IF lrHighVacuumRefReading <>0 THEN
lrVacuumSoftRatio := INT_TO_LREAL(iVacuumSoftRange) /lrHighVacuumRefReading;
END_IF


IF iAnalogInput > (32767/10) THEN
rBuffer := INT_TO_LREAL(iZeroVacuumRefValue) - INT_TO_LREAL(iAnalogInput);
ELSE
rBuffer := INT_TO_LREAL(iZeroVacuumRefValue) - 3276;  (*zero- 0*)
END_IF

IF  lrVacuumSoftRatio <>0 THEN
rVacuumPV_kPa :=rBuffer/ lrVacuumSoftRatio;
END_IF

iVacuumPV_kPa := REAL_TO_INT (rVacuumPV_kPa);

END_FUNCTION_BLOCK

// ---- FBs/B_JKS_NewFB/FBP-Instrument/fbWeberMultiFreqCtrl.TcPOU
FUNCTION_BLOCK fbWeberMultiFreqCtrl
VAR_INPUT

	bErrorReset : BOOL;
	b2550NewFirmware : BOOL;
END_VAR

VAR_IN_OUT PERSISTENT
	DSWeberGenerator : ARRAY [1..iUSGeneratorQty] OF DS_WeberGenerator;
	iStepDelaySVns: INT;
END_VAR

VAR_OUTPUT
	bFSel1OnOff :  BOOL;
	bFSel2OnOff :  BOOL;

END_VAR

VAR PERSISTENT
	ARbFreqChangeTriggerEn : ARRAY [1..iUSGeneratorQty] OF BOOL; (*Internally activate by monitor the changes of set point*)
(*	ARiPowerAnalogInput AT %I* : ARRAY [1..iUSGeneratorQty] OF INT; (*Link to Terminal*)
	ARiPowerAnalogOutput AT %Q* : ARRAY [1..iUSGeneratorQty] OF INT; (*Link to Terminal*)
*)
(**)	bFreqSwitchingPBRE: ARRAY [1..iUSGeneratorQty] OF R_TRIG;
	ARbFreqChangeMonitoringEn : ARRAY [1..iUSGeneratorQty] OF BOOL; (*Enable monitor the changes of set point*)
	ARiCurrentFreq: ARRAY [1..iUSGeneratorQty] OF INT;
	iFreqChangeStep: INT;
	iFreqChangeTriggerSet: INT;
	ARbFreqChangeTriggerEnRE: ARRAY [1..iUSGeneratorQty] OF R_TRIG;
	tStep1DelayTimer: TON;
	tStep2DelayTimer: TON;
	tStep3DelayTimer: TON;
	tStep0DelayTimer: TON;
	iGenFL: INT;
	iFreqChangeFL: INT;
END_VAR

(*Ultrasonic Start/Stop Ctrl*)
tStep0DelayTimer(IN:=iFreqChangeStep = 0 , PT:=INT_TO_TIME(iStepDelaySVns) , Q=> , ET=> );

iGenFL := 1;

	FOR iGenFL := 1 TO iUSGeneratorQty DO

				(*Min Control - Default*)
				IF DSWeberGenerator[iGenFL].IN_lrPowerToAnalogRatio <= 0 THEN
				DSWeberGenerator[iGenFL].IN_lrPowerToAnalogRatio := 327.67;
				END_IF

				(*Ultrasonic Start/Stop Ctrl*)
				IF tStep0DelayTimer.Q THEN
					IF DSWeberGenerator[iGenFL].IN_bUltrasonicStartEn THEN
					DSWeberGenerator[iGenFL].OUT_bUltrasonicOnOff := TRUE;
					ELSE
					DSWeberGenerator[iGenFL].OUT_bUltrasonicOnOff := FALSE;
					END_IF

				END_IF


				(*MultiFreq Ctrl - Change Freq via Digital Output Control*)

				(*Monitoring Start/Stop Control*)
				IF DSWeberGenerator[iGenFL].IN_bMultiFreqEn THEN
					IF DSWeberGenerator[iGenFL].DSWeberMulFreqSwitching.bFreqRange2550En AND NOT DSWeberGenerator[iGenFL].DSWeberMulFreqSwitching.bFreqRange4080120En THEN
						IF DSWeberGenerator[iGenFL].IN_iFreqSetPoint = 25 OR DSWeberGenerator[iGenFL].IN_iFreqSetPoint = 50 THEN
						ARbFreqChangeMonitoringEn[iGenFL] := TRUE;
						END_IF
					ELSIF NOT DSWeberGenerator[iGenFL].DSWeberMulFreqSwitching.bFreqRange2550En AND DSWeberGenerator[iGenFL].DSWeberMulFreqSwitching.bFreqRange4080120En THEN
						IF DSWeberGenerator[iGenFL].IN_iFreqSetPoint = 40 OR DSWeberGenerator[iGenFL].IN_iFreqSetPoint = 80 OR DSWeberGenerator[iGenFL].IN_iFreqSetPoint = 132 THEN
						ARbFreqChangeMonitoringEn[iGenFL] := TRUE;
						END_IF
					ELSE
						ARbFreqChangeMonitoringEn[iGenFL] := FALSE;
					END_IF
				ELSE
						ARbFreqChangeMonitoringEn[iGenFL] := FALSE;
				END_IF

				IF ARbFreqChangeMonitoringEn[iGenFL] THEN

					IF DSWeberGenerator[iGenFL].IN_iFreqSetPoint <> ARiCurrentFreq[iGenFL] THEN
						ARbFreqChangeTriggerEn[iGenFL] := TRUE;
					END_IF

				ELSE
					ARbFreqChangeTriggerEn[iGenFL] := FALSE;
				END_IF


				(*Analog Output*)
				IF DSWeberGenerator[iGenFL].IN_lrAnalogOutputFineTuneRatio <= 0 THEN
				DSWeberGenerator[iGenFL].IN_lrAnalogOutputFineTuneRatio := 1;
				END_IF

				IF DSWeberGenerator[iGenFL].IN_iTargetPowerPercentSetPoint <= 0 THEN
				DSWeberGenerator[iGenFL].OUT_iPowerAnalogOutput := 0;
				ELSIF DSWeberGenerator[iGenFL].IN_lrPowerToAnalogRatio <= 0 THEN
				DSWeberGenerator[iGenFL].OUT_iPowerAnalogOutput := 0;
				ELSIF (INT_TO_LREAL(DSWeberGenerator[iGenFL].IN_iTargetPowerPercentSetPoint) * DSWeberGenerator[iGenFL].IN_lrPowerToAnalogRatio) * DSWeberGenerator[iGenFL].IN_lrAnalogOutputFineTuneRatio <=32767 THEN
					DSWeberGenerator[iGenFL].OUT_iPowerAnalogOutput := LREAL_TO_INT(INT_TO_LREAL(DSWeberGenerator[iGenFL].IN_iTargetPowerPercentSetPoint) * DSWeberGenerator[iGenFL].IN_lrPowerToAnalogRatio * DSWeberGenerator[iGenFL].IN_lrAnalogOutputFineTuneRatio);
				ELSIF (INT_TO_LREAL(DSWeberGenerator[iGenFL].IN_iTargetPowerPercentSetPoint) * DSWeberGenerator[iGenFL].IN_lrPowerToAnalogRatio * DSWeberGenerator[iGenFL].IN_lrAnalogOutputFineTuneRatio) >32767 THEN
					DSWeberGenerator[iGenFL].OUT_iPowerAnalogOutput := 32767;

				ELSE
				DSWeberGenerator[iGenFL].OUT_iPowerAnalogOutput := 0;
				END_IF


				(*ActualPowerPercentageDisplay*)

				IF DSWeberGenerator[iGenFL].IN_lrAnalogInputFineTuneRatio <= 0 THEN
				DSWeberGenerator[iGenFL].IN_lrAnalogInputFineTuneRatio := 1;
				END_IF

				IF DSWeberGenerator[iGenFL].IN_iPowerAnalogInput <= 0 THEN
				DSWeberGenerator[iGenFL].OUT_iActualPowerPercentDisplay := 0;
				ELSIF DSWeberGenerator[iGenFL].IN_lrPowerToAnalogRatio <= 0 THEN
				DSWeberGenerator[iGenFL].OUT_iActualPowerPercentDisplay := 0;
				ELSIF ((INT_TO_LREAL(DSWeberGenerator[iGenFL].IN_iPowerAnalogInput) / DSWeberGenerator[iGenFL].IN_lrPowerToAnalogRatio) )* DSWeberGenerator[iGenFL].IN_lrAnalogInputFineTuneRatio <=100 THEN
					DSWeberGenerator[iGenFL].OUT_iActualPowerPercentDisplay := LREAL_TO_INT((INT_TO_LREAL(DSWeberGenerator[iGenFL].IN_iPowerAnalogInput) / DSWeberGenerator[iGenFL].IN_lrPowerToAnalogRatio) * DSWeberGenerator[iGenFL].IN_lrAnalogInputFineTuneRatio);
				ELSIF ((INT_TO_LREAL(DSWeberGenerator[iGenFL].IN_iPowerAnalogInput) / DSWeberGenerator[iGenFL].IN_lrPowerToAnalogRatio) )* DSWeberGenerator[iGenFL].IN_lrAnalogInputFineTuneRatio >100 THEN
					DSWeberGenerator[iGenFL].OUT_iActualPowerPercentDisplay := 100;

				ELSE
				DSWeberGenerator[iGenFL].OUT_iPowerAnalogOutput := 0;
				END_IF

				(*TS - FreqSwitchingPushButtonControl*)
				bFreqSwitchingPBRE[iGenFL](CLK:=DSWeberGenerator[iGenFL].DSWeberMulFreqSwitching.bFreqSwitchingPB_TS , Q=> );

				IF NOT DSWeberGenerator[iGenFL].DSWeberMulFreqSwitching.bFreqRange2550En AND NOT DSWeberGenerator[iGenFL].DSWeberMulFreqSwitching.bFreqRange4080120En THEN
				DSWeberGenerator[iGenFL].DSWeberMulFreqSwitching.iFreqOutput_TS := 0;
				ELSIF DSWeberGenerator[iGenFL].DSWeberMulFreqSwitching.bFreqRange2550En AND DSWeberGenerator[iGenFL].DSWeberMulFreqSwitching.bFreqRange4080120En THEN
				DSWeberGenerator[iGenFL].DSWeberMulFreqSwitching.iFreqOutput_TS := 0;


				ELSIF DSWeberGenerator[iGenFL].DSWeberMulFreqSwitching.bFreqRange2550En AND NOT DSWeberGenerator[iGenFL].DSWeberMulFreqSwitching.bFreqRange4080120En THEN

					IF DSWeberGenerator[iGenFL].DSWeberMulFreqSwitching.iFreqOutput_TS <> 25 AND DSWeberGenerator[iGenFL].DSWeberMulFreqSwitching.iFreqOutput_TS <> 50 THEN
					DSWeberGenerator[iGenFL].DSWeberMulFreqSwitching.iFreqOutput_TS := 25;
					END_IF

					IF bFreqSwitchingPBRE[iGenFL].Q THEN
						IF DSWeberGenerator[iGenFL].DSWeberMulFreqSwitching.iFreqOutput_TS = 25 THEN
						DSWeberGenerator[iGenFL].DSWeberMulFreqSwitching.iFreqOutput_TS := 50;
						ELSIF DSWeberGenerator[iGenFL].DSWeberMulFreqSwitching.iFreqOutput_TS = 50 THEN
						DSWeberGenerator[iGenFL].DSWeberMulFreqSwitching.iFreqOutput_TS := 25;
						END_IF
					END_IF


				ELSIF NOT DSWeberGenerator[iGenFL].DSWeberMulFreqSwitching.bFreqRange2550En AND DSWeberGenerator[iGenFL].DSWeberMulFreqSwitching.bFreqRange4080120En THEN

					IF DSWeberGenerator[iGenFL].DSWeberMulFreqSwitching.iFreqOutput_TS <> 40 AND DSWeberGenerator[iGenFL].DSWeberMulFreqSwitching.iFreqOutput_TS <> 80 AND DSWeberGenerator[iGenFL].DSWeberMulFreqSwitching.iFreqOutput_TS <> 132  THEN
					DSWeberGenerator[iGenFL].DSWeberMulFreqSwitching.iFreqOutput_TS := 40;
					END_IF

					IF bFreqSwitchingPBRE[iGenFL].Q AND NOT DSWeberGenerator[iGenFL].DSWeberMulFreqSwitching.bDisableMultiFreq80kHz THEN
						IF DSWeberGenerator[iGenFL].DSWeberMulFreqSwitching.iFreqOutput_TS = 40 THEN
						DSWeberGenerator[iGenFL].DSWeberMulFreqSwitching.iFreqOutput_TS := 80;
						ELSIF DSWeberGenerator[iGenFL].DSWeberMulFreqSwitching.iFreqOutput_TS = 80 THEN
						DSWeberGenerator[iGenFL].DSWeberMulFreqSwitching.iFreqOutput_TS := 132;
						ELSIF DSWeberGenerator[iGenFL].DSWeberMulFreqSwitching.iFreqOutput_TS = 132 THEN
						DSWeberGenerator[iGenFL].DSWeberMulFreqSwitching.iFreqOutput_TS := 40;
						END_IF

					ELSIF bFreqSwitchingPBRE[iGenFL].Q AND DSWeberGenerator[iGenFL].DSWeberMulFreqSwitching.bDisableMultiFreq80kHz THEN
						IF DSWeberGenerator[iGenFL].DSWeberMulFreqSwitching.iFreqOutput_TS = 40 THEN
						DSWeberGenerator[iGenFL].DSWeberMulFreqSwitching.iFreqOutput_TS := 132;
						ELSIF DSWeberGenerator[iGenFL].DSWeberMulFreqSwitching.iFreqOutput_TS = 132 THEN
						DSWeberGenerator[iGenFL].DSWeberMulFreqSwitching.iFreqOutput_TS := 40;
						END_IF

					END_IF

				END_IF

	END_FOR



(*Seperate FL to control*)

IF iFreqChangeStep = 0 THEN
iFreqChangeFL := 1;
	FOR iFreqChangeFL := 1 TO iUSGeneratorQty DO

		IF ARbFreqChangeTriggerEn[iFreqChangeFL] THEN
		iFreqChangeStep := 1;
		iFreqChangeTriggerSet := iFreqChangeFL;
		iFreqChangeFL := iUSGeneratorQty +1;
		END_IF
	END_FOR
END_IF

(*******************************************************************************************)






(*Freq Change Start*)

IF iStepDelaySVns < 300 THEN
iStepDelaySVns := 300;
END_IF


(*Freq Change Sequence Start*)
tStep1DelayTimer(IN:=iFreqChangeStep=1 , PT:=INT_TO_TIME(iStepDelaySVns) , Q=> , ET=> );
tStep2DelayTimer(IN:=iFreqChangeStep=2 , PT:=INT_TO_TIME(iStepDelaySVns) , Q=> , ET=> );
tStep3DelayTimer(IN:=iFreqChangeStep=3 , PT:=INT_TO_TIME(iStepDelaySVns) , Q=> , ET=> );

CASE iFreqChangeStep OF
0:
	bFSel1OnOff := FALSE;
	bFSel2OnOff := FALSE;


1:
DSWeberGenerator[iFreqChangeTriggerSet].OUT_bUltrasonicOnOff := FALSE;

IF DSWeberGenerator[iFreqChangeTriggerSet].DSWeberMulFreqSwitching.bFreqRange2550En AND NOT b2550NewFirmware THEN

	IF DSWeberGenerator[iFreqChangeTriggerSet].IN_iFreqSetPoint = 25 THEN
	bFSel1OnOff := TRUE;
	bFSel2OnOff := FALSE;
	ELSIF DSWeberGenerator[iFreqChangeTriggerSet].IN_iFreqSetPoint = 50 THEN
	bFSel1OnOff := FALSE;
	bFSel2OnOff := TRUE;
	ELSIF DSWeberGenerator[iFreqChangeTriggerSet].IN_iFreqSetPoint = 0 THEN
	bFSel1OnOff := FALSE;
	bFSel2OnOff := FALSE;
	ELSE
	bFSel1OnOff := FALSE;
	bFSel2OnOff := FALSE;
	iFreqChangeStep := 4;
	END_IF

ELSIF DSWeberGenerator[iFreqChangeTriggerSet].DSWeberMulFreqSwitching.bFreqRange2550En AND b2550NewFirmware THEN

	IF DSWeberGenerator[iFreqChangeTriggerSet].IN_iFreqSetPoint = 25 THEN
	bFSel1OnOff := TRUE;
	bFSel2OnOff := TRUE;
	ELSIF DSWeberGenerator[iFreqChangeTriggerSet].IN_iFreqSetPoint = 50 THEN
	bFSel1OnOff := FALSE;
	bFSel2OnOff := TRUE;
	ELSIF DSWeberGenerator[iFreqChangeTriggerSet].IN_iFreqSetPoint = 0 THEN
	bFSel1OnOff := FALSE;
	bFSel2OnOff := FALSE;
	ELSE
	bFSel1OnOff := FALSE;
	bFSel2OnOff := FALSE;
	iFreqChangeStep := 4;
	END_IF

END_IF

IF DSWeberGenerator[iFreqChangeTriggerSet].DSWeberMulFreqSwitching.bFreqRange4080120En THEN

	IF NOT DSWeberGenerator[iFreqChangeTriggerSet].DSWeberMulFreqSwitching.bDisableMultiFreq80kHz THEN

			IF DSWeberGenerator[iFreqChangeTriggerSet].IN_iFreqSetPoint = 40 THEN
			bFSel1OnOff := TRUE;
			bFSel2OnOff := TRUE;
			ELSIF DSWeberGenerator[iFreqChangeTriggerSet].IN_iFreqSetPoint = 80 THEN
			bFSel1OnOff := FALSE;
			bFSel2OnOff := TRUE;
			ELSIF DSWeberGenerator[iFreqChangeTriggerSet].IN_iFreqSetPoint = 132 THEN
			bFSel1OnOff := TRUE;
			bFSel2OnOff := FALSE;
			ELSIF DSWeberGenerator[iFreqChangeTriggerSet].IN_iFreqSetPoint = 0 THEN
			bFSel1OnOff := FALSE;
			bFSel2OnOff := FALSE;
			ELSE
			bFSel1OnOff := FALSE;
			bFSel2OnOff := FALSE;
			iFreqChangeStep := 4;
			END_IF
	ELSE

			IF DSWeberGenerator[iFreqChangeTriggerSet].IN_iFreqSetPoint = 40 THEN
			bFSel1OnOff := TRUE;
			bFSel2OnOff := FALSE;
			ELSIF DSWeberGenerator[iFreqChangeTriggerSet].IN_iFreqSetPoint = 132 THEN
			bFSel1OnOff := FALSE;
			bFSel2OnOff := TRUE;
			ELSIF DSWeberGenerator[iFreqChangeTriggerSet].IN_iFreqSetPoint = 0 THEN
			bFSel1OnOff := FALSE;
			bFSel2OnOff := FALSE;
			ELSE
			bFSel1OnOff := FALSE;
			bFSel2OnOff := FALSE;
			iFreqChangeStep := 4;
			END_IF
	END_IF



END_IF


IF tStep1DelayTimer.Q THEN
iFreqChangeStep := 2;
END_IF

2:
IF DSWeberGenerator[iFreqChangeTriggerSet].IN_iFreqSetPoint <> 0 THEN
DSWeberGenerator[iFreqChangeTriggerSet].OUT_bUltrasonicOnOff := TRUE;
ELSE
DSWeberGenerator[iFreqChangeTriggerSet].OUT_bUltrasonicOnOff := FALSE;
END_IF

IF tStep2DelayTimer.Q THEN
iFreqChangeStep := 3;
END_IF

3:
DSWeberGenerator[iFreqChangeTriggerSet].OUT_bUltrasonicOnOff := FALSE;
bFSel1OnOff := FALSE;
bFSel2OnOff := FALSE;

IF tStep3DelayTimer.Q THEN
iFreqChangeStep := 0;
ARbFreqChangeTriggerEn[iFreqChangeTriggerSet] := FALSE;
ARiCurrentFreq[iFreqChangeTriggerSet] := DSWeberGenerator[iFreqChangeTriggerSet].IN_iFreqSetPoint;
END_IF

4: (*Error*)
DSWeberGenerator[iFreqChangeTriggerSet].OUT_bFreqSetPointError := TRUE;
iFreqChangeStep := 5;


5: (*Error - Waiting Reset*)
IF bErrorReset THEN
DSWeberGenerator[iFreqChangeTriggerSet].OUT_bFreqSetPointError := FALSE;
iFreqChangeStep := 0;
ARbFreqChangeTriggerEn[iFreqChangeTriggerSet] := FALSE;
ARiCurrentFreq[iFreqChangeTriggerSet] := DSWeberGenerator[iFreqChangeTriggerSet].IN_iFreqSetPoint;
END_IF

END_CASE

END_FUNCTION_BLOCK

// ---- FBs/B_JKS_NewFB/FBP-Instrument/fbBrensonMultiFreqCtrl.TcPOU
FUNCTION_BLOCK fbBrensonMultiFreqCtrl
VAR_INPUT

	bErrorReset : BOOL;
	b2550NewFirmware : BOOL;
END_VAR

VAR_IN_OUT PERSISTENT
	DSBrensonGenerator : ARRAY [1..iUSGeneratorQty] OF DS_BrensonGenerator;
	iStepDelaySVns: INT;
END_VAR

VAR_OUTPUT
	bFSel1OnOff :  BOOL;
	bFSel2OnOff :  BOOL;

END_VAR

VAR PERSISTENT
	ARbFreqChangeTriggerEn : ARRAY [1..iUSGeneratorQty] OF BOOL; (*Internally activate by monitor the changes of set point*)
(*	ARiPowerAnalogInput AT %I* : ARRAY [1..iUSGeneratorQty] OF INT; (*Link to Terminal*)
	ARiPowerAnalogOutput AT %Q* : ARRAY [1..iUSGeneratorQty] OF INT; (*Link to Terminal*)
*)
(**)	bFreqSwitchingPBRE: ARRAY [1..iUSGeneratorQty] OF R_TRIG;
	ARbFreqChangeMonitoringEn : ARRAY [1..iUSGeneratorQty] OF BOOL; (*Enable monitor the changes of set point*)
	ARiCurrentFreq: ARRAY [1..iUSGeneratorQty] OF INT;
	iFreqChangeStep: INT;
	iFreqChangeTriggerSet: INT;
	ARbFreqChangeTriggerEnRE: ARRAY [1..iUSGeneratorQty] OF R_TRIG;
	tStep1DelayTimer: TON;
	tStep2DelayTimer: TON;
	tStep3DelayTimer: TON;
	tStep0DelayTimer: TON;
	iGenFL: INT;
	iFreqChangeFL: INT;
END_VAR

(*Ultrasonic Start/Stop Ctrl*)
tStep0DelayTimer(IN:=iFreqChangeStep = 0 , PT:=INT_TO_TIME(iStepDelaySVns) , Q=> , ET=> );

iGenFL := 1;

	FOR iGenFL := 1 TO iUSGeneratorQty DO

				(*Min Control - Default*)
				IF DSBrensonGenerator[iGenFL].IN_lrPowerToAnalogRatio <= 0 THEN
				DSBrensonGenerator[iGenFL].IN_lrPowerToAnalogRatio := 327.67;
				END_IF

				(*Ultrasonic Start/Stop Ctrl*)
				IF tStep0DelayTimer.Q THEN
					IF DSBrensonGenerator[iGenFL].IN_bUltrasonicStartEn THEN
					DSBrensonGenerator[iGenFL].OUT_bUltrasonicOnOff := TRUE;
					ELSE
					DSBrensonGenerator[iGenFL].OUT_bUltrasonicOnOff := FALSE;
					END_IF

				END_IF


				(*MultiFreq Ctrl - Change Freq via Digital Output Control*)

				(*Monitoring Start/Stop Control*)
				IF DSBrensonGenerator[iGenFL].IN_bMultiFreqEn THEN
					IF DSBrensonGenerator[iGenFL].DSBrensonMulFreqSwitching.bFreqRange2550En AND NOT DSBrensonGenerator[iGenFL].DSBrensonMulFreqSwitching.bFreqRange4080120En THEN
						IF DSBrensonGenerator[iGenFL].IN_iFreqSetPoint = 25 OR DSBrensonGenerator[iGenFL].IN_iFreqSetPoint = 50 THEN
						ARbFreqChangeMonitoringEn[iGenFL] := TRUE;
						END_IF
					ELSIF NOT DSBrensonGenerator[iGenFL].DSBrensonMulFreqSwitching.bFreqRange2550En AND DSBrensonGenerator[iGenFL].DSBrensonMulFreqSwitching.bFreqRange4080120En THEN
						IF DSBrensonGenerator[iGenFL].IN_iFreqSetPoint = 40 OR DSBrensonGenerator[iGenFL].IN_iFreqSetPoint = 80 OR DSBrensonGenerator[iGenFL].IN_iFreqSetPoint = 120 THEN
						ARbFreqChangeMonitoringEn[iGenFL] := TRUE;
						END_IF
					ELSE
						ARbFreqChangeMonitoringEn[iGenFL] := FALSE;
					END_IF
				ELSE
						ARbFreqChangeMonitoringEn[iGenFL] := FALSE;
				END_IF

				IF ARbFreqChangeMonitoringEn[iGenFL] THEN

					IF DSBrensonGenerator[iGenFL].IN_iFreqSetPoint <> ARiCurrentFreq[iGenFL] THEN
						ARbFreqChangeTriggerEn[iGenFL] := TRUE;
					END_IF

				ELSE
					ARbFreqChangeTriggerEn[iGenFL] := FALSE;
				END_IF


				(*Analog Output*)
				IF DSBrensonGenerator[iGenFL].IN_lrAnalogOutputFineTuneRatio <= 0 THEN
				DSBrensonGenerator[iGenFL].IN_lrAnalogOutputFineTuneRatio := 1;
				END_IF

				IF DSBrensonGenerator[iGenFL].IN_iTargetPowerPercentSetPoint <= 0 THEN
				DSBrensonGenerator[iGenFL].OUT_iPowerAnalogOutput := 0;
				ELSIF DSBrensonGenerator[iGenFL].IN_lrPowerToAnalogRatio <= 0 THEN
				DSBrensonGenerator[iGenFL].OUT_iPowerAnalogOutput := 0;
				ELSIF (INT_TO_LREAL(DSBrensonGenerator[iGenFL].IN_iTargetPowerPercentSetPoint) * DSBrensonGenerator[iGenFL].IN_lrPowerToAnalogRatio) * DSBrensonGenerator[iGenFL].IN_lrAnalogOutputFineTuneRatio <=32767 THEN
					DSBrensonGenerator[iGenFL].OUT_iPowerAnalogOutput := LREAL_TO_INT(INT_TO_LREAL(DSBrensonGenerator[iGenFL].IN_iTargetPowerPercentSetPoint) * DSBrensonGenerator[iGenFL].IN_lrPowerToAnalogRatio * DSBrensonGenerator[iGenFL].IN_lrAnalogOutputFineTuneRatio);
				ELSIF (INT_TO_LREAL(DSBrensonGenerator[iGenFL].IN_iTargetPowerPercentSetPoint) * DSBrensonGenerator[iGenFL].IN_lrPowerToAnalogRatio * DSBrensonGenerator[iGenFL].IN_lrAnalogOutputFineTuneRatio) >32767 THEN
					DSBrensonGenerator[iGenFL].OUT_iPowerAnalogOutput := 32767;

				ELSE
				DSBrensonGenerator[iGenFL].OUT_iPowerAnalogOutput := 0;
				END_IF


				(*ActualPowerPercentageDisplay*)

				IF DSBrensonGenerator[iGenFL].IN_lrAnalogInputFineTuneRatio <= 0 THEN
				DSBrensonGenerator[iGenFL].IN_lrAnalogInputFineTuneRatio := 1;
				END_IF

				IF DSBrensonGenerator[iGenFL].IN_iPowerAnalogInput <= 0 THEN
				DSBrensonGenerator[iGenFL].OUT_iActualPowerPercentDisplay := 0;
				ELSIF DSBrensonGenerator[iGenFL].IN_lrPowerToAnalogRatio <= 0 THEN
				DSBrensonGenerator[iGenFL].OUT_iActualPowerPercentDisplay := 0;
				ELSIF ((INT_TO_LREAL(DSBrensonGenerator[iGenFL].IN_iPowerAnalogInput) / DSBrensonGenerator[iGenFL].IN_lrPowerToAnalogRatio) )* DSBrensonGenerator[iGenFL].IN_lrAnalogInputFineTuneRatio <=100 THEN
					DSBrensonGenerator[iGenFL].OUT_iActualPowerPercentDisplay := LREAL_TO_INT((INT_TO_LREAL(DSBrensonGenerator[iGenFL].IN_iPowerAnalogInput) / DSBrensonGenerator[iGenFL].IN_lrPowerToAnalogRatio) * DSBrensonGenerator[iGenFL].IN_lrAnalogInputFineTuneRatio);
				ELSIF ((INT_TO_LREAL(DSBrensonGenerator[iGenFL].IN_iPowerAnalogInput) / DSBrensonGenerator[iGenFL].IN_lrPowerToAnalogRatio) )* DSBrensonGenerator[iGenFL].IN_lrAnalogInputFineTuneRatio >100 THEN
					DSBrensonGenerator[iGenFL].OUT_iActualPowerPercentDisplay := 100;

				ELSE
				DSBrensonGenerator[iGenFL].OUT_iPowerAnalogOutput := 0;
				END_IF

				(*TS - FreqSwitchingPushButtonControl*)
				bFreqSwitchingPBRE[iGenFL](CLK:=DSBrensonGenerator[iGenFL].DSBrensonMulFreqSwitching.bFreqSwitchingPB_TS , Q=> );

				IF NOT DSBrensonGenerator[iGenFL].DSBrensonMulFreqSwitching.bFreqRange2550En AND NOT DSBrensonGenerator[iGenFL].DSBrensonMulFreqSwitching.bFreqRange4080120En THEN
				DSBrensonGenerator[iGenFL].DSBrensonMulFreqSwitching.iFreqOutput_TS := 0;
				ELSIF DSBrensonGenerator[iGenFL].DSBrensonMulFreqSwitching.bFreqRange2550En AND DSBrensonGenerator[iGenFL].DSBrensonMulFreqSwitching.bFreqRange4080120En THEN
				DSBrensonGenerator[iGenFL].DSBrensonMulFreqSwitching.iFreqOutput_TS := 0;


				ELSIF DSBrensonGenerator[iGenFL].DSBrensonMulFreqSwitching.bFreqRange2550En AND NOT DSBrensonGenerator[iGenFL].DSBrensonMulFreqSwitching.bFreqRange4080120En THEN

					IF DSBrensonGenerator[iGenFL].DSBrensonMulFreqSwitching.iFreqOutput_TS <> 25 AND DSBrensonGenerator[iGenFL].DSBrensonMulFreqSwitching.iFreqOutput_TS <> 50 THEN
					DSBrensonGenerator[iGenFL].DSBrensonMulFreqSwitching.iFreqOutput_TS := 25;
					END_IF

					IF bFreqSwitchingPBRE[iGenFL].Q THEN
						IF DSBrensonGenerator[iGenFL].DSBrensonMulFreqSwitching.iFreqOutput_TS = 25 THEN
						DSBrensonGenerator[iGenFL].DSBrensonMulFreqSwitching.iFreqOutput_TS := 50;
						ELSIF DSBrensonGenerator[iGenFL].DSBrensonMulFreqSwitching.iFreqOutput_TS = 50 THEN
						DSBrensonGenerator[iGenFL].DSBrensonMulFreqSwitching.iFreqOutput_TS := 25;
						END_IF
					END_IF


				ELSIF NOT DSBrensonGenerator[iGenFL].DSBrensonMulFreqSwitching.bFreqRange2550En AND DSBrensonGenerator[iGenFL].DSBrensonMulFreqSwitching.bFreqRange4080120En THEN

					IF DSBrensonGenerator[iGenFL].DSBrensonMulFreqSwitching.iFreqOutput_TS <> 40 AND DSBrensonGenerator[iGenFL].DSBrensonMulFreqSwitching.iFreqOutput_TS <> 80 AND DSBrensonGenerator[iGenFL].DSBrensonMulFreqSwitching.iFreqOutput_TS <> 120  THEN
					DSBrensonGenerator[iGenFL].DSBrensonMulFreqSwitching.iFreqOutput_TS := 40;
					END_IF

					IF bFreqSwitchingPBRE[iGenFL].Q AND NOT DSBrensonGenerator[iGenFL].DSBrensonMulFreqSwitching.bDisableMultiFreq80kHz THEN
						IF DSBrensonGenerator[iGenFL].DSBrensonMulFreqSwitching.iFreqOutput_TS = 40 THEN
						DSBrensonGenerator[iGenFL].DSBrensonMulFreqSwitching.iFreqOutput_TS := 80;
						ELSIF DSBrensonGenerator[iGenFL].DSBrensonMulFreqSwitching.iFreqOutput_TS = 80 THEN
						DSBrensonGenerator[iGenFL].DSBrensonMulFreqSwitching.iFreqOutput_TS := 120;
						ELSIF DSBrensonGenerator[iGenFL].DSBrensonMulFreqSwitching.iFreqOutput_TS = 120 THEN
						DSBrensonGenerator[iGenFL].DSBrensonMulFreqSwitching.iFreqOutput_TS := 40;
						END_IF

					ELSIF bFreqSwitchingPBRE[iGenFL].Q AND DSBrensonGenerator[iGenFL].DSBrensonMulFreqSwitching.bDisableMultiFreq80kHz THEN
						IF DSBrensonGenerator[iGenFL].DSBrensonMulFreqSwitching.iFreqOutput_TS = 40 THEN
						DSBrensonGenerator[iGenFL].DSBrensonMulFreqSwitching.iFreqOutput_TS := 120;
						ELSIF DSBrensonGenerator[iGenFL].DSBrensonMulFreqSwitching.iFreqOutput_TS = 120 THEN
						DSBrensonGenerator[iGenFL].DSBrensonMulFreqSwitching.iFreqOutput_TS := 40;
						END_IF

					END_IF

				END_IF

	END_FOR



(*Seperate FL to control*)

IF iFreqChangeStep = 0 THEN
iFreqChangeFL := 1;
	FOR iFreqChangeFL := 1 TO iUSGeneratorQty DO

		IF ARbFreqChangeTriggerEn[iFreqChangeFL] THEN
		iFreqChangeStep := 1;
		iFreqChangeTriggerSet := iFreqChangeFL;
		iFreqChangeFL := iUSGeneratorQty +1;
		END_IF
	END_FOR
END_IF

(*******************************************************************************************)






(*Freq Change Start*)

IF iStepDelaySVns < 300 THEN
iStepDelaySVns := 300;
END_IF


(*Freq Change Sequence Start*)
tStep1DelayTimer(IN:=iFreqChangeStep=1 , PT:=INT_TO_TIME(iStepDelaySVns) , Q=> , ET=> );
tStep2DelayTimer(IN:=iFreqChangeStep=2 , PT:=INT_TO_TIME(iStepDelaySVns) , Q=> , ET=> );
tStep3DelayTimer(IN:=iFreqChangeStep=3 , PT:=INT_TO_TIME(iStepDelaySVns) , Q=> , ET=> );

CASE iFreqChangeStep OF
0:
	bFSel1OnOff := FALSE;
	bFSel2OnOff := FALSE;


1:
DSBrensonGenerator[iFreqChangeTriggerSet].OUT_bUltrasonicOnOff := FALSE;

IF DSBrensonGenerator[iFreqChangeTriggerSet].DSBrensonMulFreqSwitching.bFreqRange2550En AND NOT b2550NewFirmware THEN

	IF DSBrensonGenerator[iFreqChangeTriggerSet].IN_iFreqSetPoint = 25 THEN
	bFSel1OnOff := TRUE;
	bFSel2OnOff := FALSE;
	ELSIF DSBrensonGenerator[iFreqChangeTriggerSet].IN_iFreqSetPoint = 50 THEN
	bFSel1OnOff := FALSE;
	bFSel2OnOff := TRUE;
	ELSIF DSBrensonGenerator[iFreqChangeTriggerSet].IN_iFreqSetPoint = 0 THEN
	bFSel1OnOff := FALSE;
	bFSel2OnOff := FALSE;
	ELSE
	bFSel1OnOff := FALSE;
	bFSel2OnOff := FALSE;
	iFreqChangeStep := 4;
	END_IF

ELSIF DSBrensonGenerator[iFreqChangeTriggerSet].DSBrensonMulFreqSwitching.bFreqRange2550En AND b2550NewFirmware THEN

	IF DSBrensonGenerator[iFreqChangeTriggerSet].IN_iFreqSetPoint = 25 THEN
	bFSel1OnOff := TRUE;
	bFSel2OnOff := TRUE;
	ELSIF DSBrensonGenerator[iFreqChangeTriggerSet].IN_iFreqSetPoint = 50 THEN
	bFSel1OnOff := FALSE;
	bFSel2OnOff := TRUE;
	ELSIF DSBrensonGenerator[iFreqChangeTriggerSet].IN_iFreqSetPoint = 0 THEN
	bFSel1OnOff := FALSE;
	bFSel2OnOff := FALSE;
	ELSE
	bFSel1OnOff := FALSE;
	bFSel2OnOff := FALSE;
	iFreqChangeStep := 4;
	END_IF

END_IF

IF DSBrensonGenerator[iFreqChangeTriggerSet].DSBrensonMulFreqSwitching.bFreqRange4080120En THEN

	IF NOT DSBrensonGenerator[iFreqChangeTriggerSet].DSBrensonMulFreqSwitching.bDisableMultiFreq80kHz THEN

			IF DSBrensonGenerator[iFreqChangeTriggerSet].IN_iFreqSetPoint = 40 THEN
			bFSel1OnOff := TRUE;
			bFSel2OnOff := TRUE;
			ELSIF DSBrensonGenerator[iFreqChangeTriggerSet].IN_iFreqSetPoint = 80 THEN
			bFSel1OnOff := FALSE;
			bFSel2OnOff := TRUE;
			ELSIF DSBrensonGenerator[iFreqChangeTriggerSet].IN_iFreqSetPoint = 120 THEN
			bFSel1OnOff := TRUE;
			bFSel2OnOff := FALSE;
			ELSIF DSBrensonGenerator[iFreqChangeTriggerSet].IN_iFreqSetPoint = 0 THEN
			bFSel1OnOff := FALSE;
			bFSel2OnOff := FALSE;
			ELSE
			bFSel1OnOff := FALSE;
			bFSel2OnOff := FALSE;
			iFreqChangeStep := 4;
			END_IF
	ELSE

			IF DSBrensonGenerator[iFreqChangeTriggerSet].IN_iFreqSetPoint = 40 THEN
			bFSel1OnOff := TRUE;
			bFSel2OnOff := FALSE;
			ELSIF DSBrensonGenerator[iFreqChangeTriggerSet].IN_iFreqSetPoint = 120 THEN
			bFSel1OnOff := FALSE;
			bFSel2OnOff := TRUE;
			ELSIF DSBrensonGenerator[iFreqChangeTriggerSet].IN_iFreqSetPoint = 0 THEN
			bFSel1OnOff := FALSE;
			bFSel2OnOff := FALSE;
			ELSE
			bFSel1OnOff := FALSE;
			bFSel2OnOff := FALSE;
			iFreqChangeStep := 4;
			END_IF
	END_IF



END_IF


IF tStep1DelayTimer.Q THEN
iFreqChangeStep := 2;
END_IF

2:
IF DSBrensonGenerator[iFreqChangeTriggerSet].IN_iFreqSetPoint <> 0 THEN
DSBrensonGenerator[iFreqChangeTriggerSet].OUT_bUltrasonicOnOff := TRUE;
ELSE
DSBrensonGenerator[iFreqChangeTriggerSet].OUT_bUltrasonicOnOff := FALSE;
END_IF

IF tStep2DelayTimer.Q THEN
iFreqChangeStep := 3;
END_IF

3:
DSBrensonGenerator[iFreqChangeTriggerSet].OUT_bUltrasonicOnOff := FALSE;
bFSel1OnOff := FALSE;
bFSel2OnOff := FALSE;

IF tStep3DelayTimer.Q THEN
iFreqChangeStep := 0;
ARbFreqChangeTriggerEn[iFreqChangeTriggerSet] := FALSE;
ARiCurrentFreq[iFreqChangeTriggerSet] := DSBrensonGenerator[iFreqChangeTriggerSet].IN_iFreqSetPoint;
END_IF

4: (*Error*)
DSBrensonGenerator[iFreqChangeTriggerSet].OUT_bFreqSetPointError := TRUE;
iFreqChangeStep := 5;


5: (*Error - Waiting Reset*)
IF bErrorReset THEN
DSBrensonGenerator[iFreqChangeTriggerSet].OUT_bFreqSetPointError := FALSE;
iFreqChangeStep := 0;
ARbFreqChangeTriggerEn[iFreqChangeTriggerSet] := FALSE;
ARiCurrentFreq[iFreqChangeTriggerSet] := DSBrensonGenerator[iFreqChangeTriggerSet].IN_iFreqSetPoint;
END_IF

END_CASE

END_FUNCTION_BLOCK

// ---- FBs/B_JKS_CustomFB/fbBarcodeCtrl/fbBarcodeTracer.TcPOU
FUNCTION_BLOCK fbBarcodeTracer
VAR_INPUT
	bTracerST : BOOL;
	sTargetBarcode : STRING;
	AR99sBarCodeRaw : ARRAY [0..iProductRecipeArrayQty] OF STRING;
	AR99sBarcodeDescrip	: ARRAY [0..iProductRecipeArrayQty] OF STRING;


END_VAR
VAR_OUTPUT

	bBarcodeTraceSuccess : BOOL;
	bBarcodeTraceFail : BOOL;
	iBarcodeInRecipeNo : INT;
	sBarcodeInDescrip	: STRING;
END_VAR
VAR
	i: INT;
	TracerRE : R_TRIG;

	sBuffer: STRING;
	STEP: INT;
END_VAR

TracerRE(CLK:=bTracerST,Q=>);

IF NOT bTracerST THEN
	bBarcodeTraceSuccess := FALSE;
	bBarcodeTraceFail := FALSE;
	iBarcodeInRecipeNo := 0;
	i := 1;
END_IF

IF bTracerST AND sTargetBarcode <> '' (*AND sTargetBarcode <> sBuffer*) THEN

		(*sBuffer := sTargetBarcode;*)
		FOR i := 1 TO 99 DO

		IF sTargetBarcode = AR99sBarCodeRaw[i] THEN
		sBarcodeInDescrip := AR99sBarcodeDescrip[i];
		iBarcodeInRecipeNo := i;
		bBarcodeTraceSuccess := TRUE;
		(*bBarcodeTraceFail := FALSE;*)
		i := 100;
		(*ELSE
		bBarcodeTraceFail := TRUE;
		bBarcodeTraceSuccess := FALSE;*)
		END_IF

		END_FOR

END_IF
IF (i > 99 AND bTracerST AND NOT bBarcodeTraceSuccess) (*OR (sTargetBarcode = '')*) THEN
bBarcodeTraceFail := TRUE;
ELSE
bBarcodeTraceFail := FALSE;
END_IF

END_FUNCTION_BLOCK

// ---- FBs/B_JKS_CustomFB/fbBarcodeCtrl/fbPreSuffixEliminator.TcPOU
FUNCTION_BLOCK fbPreSuffixEliminator
VAR_INPUT
	bEN									: BOOL;
	bPrefixEliminatorEN					: BOOL;
	bSuffixEliminatorEN					: BOOL;
	sData								: STRING;
	sPrefix								: STRING (*:='$02'*);
	sSuffix								:STRING;
	iLengthAfterPrefix						: INT;
	iLengthBeforeSuffix					: INT;

END_VAR
VAR_OUTPUT

	sPrefixEliminatorResult					: STRING;
	sSuffixEliminatorResult					: STRING;
	sPreSuffixEliminatorResult				: STRING;
	sNoneEliminatorReseult				: STRING;

END_VAR
VAR
	iBCPrefixFound						: INT;
	iBCSuffixFound						: INT;
	sIntPrefixEliminatorResult				: STRING;
END_VAR

(*Prefix Eliminator*)
IF bEN AND bPrefixEliminatorEN AND NOT bSuffixEliminatorEN THEN

sSuffixEliminatorResult := '';
sPreSuffixEliminatorResult := '';

iBCPrefixFound:=FIND(sData, sPrefix);
sPrefixEliminatorResult:=RIGHT(sData, iBCPrefixFound+iLengthAfterPrefix);

END_IF

(*Suffix Eliminator*)
IF bEN AND bSuffixEliminatorEN AND NOT bPrefixEliminatorEN THEN

sPrefixEliminatorResult := '';
sPreSuffixEliminatorResult := '';


iBCSuffixFound:=FIND(sData, sSuffix);
sSuffixEliminatorResult:=LEFT(sData, iBCSuffixFound-iLengthBeforeSuffix);

END_IF



IF bEN AND bSuffixEliminatorEN AND bPrefixEliminatorEN THEN

sPrefixEliminatorResult := '';
sSuffixEliminatorResult := '';

iBCPrefixFound:=FIND(sData, sPrefix);
sIntPrefixEliminatorResult:=RIGHT(sData, iBCPrefixFound+iLengthAfterPrefix);


iBCSuffixFound:=FIND(sIntPrefixEliminatorResult, sSuffix);
sPreSuffixEliminatorResult:=LEFT(sIntPrefixEliminatorResult, iBCSuffixFound-iLengthBeforeSuffix);

END_IF



IF bEN AND NOT bSuffixEliminatorEN AND NOT bPrefixEliminatorEN THEN

sNoneEliminatorReseult:=sData;

END_IF

END_FUNCTION_BLOCK

// ---- FBs/B_JKS_CustomFB/fbBarcodeCtrl/fbBarcodeSorting_10ML5575.TcPOU
FUNCTION_BLOCK fbBarcodeSorting_10ML5575
VAR_INPUT
	bEN : BOOL;
	bBarcodeTracerInvalidFlag : BOOL;
	bConfirmPB : BOOL;

	ARbBarcodeStorageEnable : ARRAY [0..10] OF BOOL;

END_VAR
VAR_IN_OUT
	sBarcodeInputFromScanner : STRING;
	ARbHMIBarcodeScanEn : ARRAY [0..10] OF BOOL;
	ARsHMIBarcodeData_ScanIn : ARRAY [0..10] OF STRING(50);


	(*Result for Out after Confirm button press*)
	ARsBarcodeData_LdBasketInfo : ARRAY [0..10] OF STRING(50);

END_VAR

VAR_OUTPUT
	bBarcodeScanEnableFlag : BOOL;
	bConfirmReadyFlag : BOOL;
END_VAR
VAR

	ARbHMIBarcodeScanEnRE: ARRAY [0..10] OF R_TRIG;
	iREFL: INT;
	iREFL2: INT;
	iScanFL: INT;
	iConfirmFL: INT;
	ARsHMIBarcodeData_Empty : ARRAY [0..10] OF STRING(50);
	bConfirmPBRE: R_TRIG;
END_VAR

bConfirmPBRE(CLK:= bConfirmPB, Q=> );


iREFL := 1;
FOR iREFL := 1 TO 10 DO
	IF iREFL >= 1 AND iREFL <= 10 THEN
		ARbHMIBarcodeScanEnRE[iREFL](CLK:=ARbHMIBarcodeScanEn[iREFL] , Q=> );

		IF ARbHMIBarcodeScanEnRE[iREFL].Q THEN
			iREFL2 := 1;

			FOR iREFL2 := 1 TO 10 DO
				ARbHMIBarcodeScanEn[iREFL2] := FALSE;
			END_FOR

			ARbHMIBarcodeScanEn[iREFL] := TRUE;
			bBarcodeScanEnableFlag := TRUE;
		END_IF
	END_IF

END_FOR

iScanFL := 1;
FOR iScanFL := 1 TO 10 DO
	IF iScanFL >= 1 AND iScanFL <= 10 THEN


		IF ARbBarcodeStorageEnable[iScanFL] (*AND ARbHMIBarcodeScanEn[iScanFL] *) AND sBarcodeInputFromScanner <> '' THEN
			ARsHMIBarcodeData_ScanIn[iScanFL]	:= sBarcodeInputFromScanner;
			bBarcodeScanEnableFlag 				:= FALSE;
			ARbHMIBarcodeScanEn[iScanFL] 		:= FALSE;
			(*sBarcodeInputFromScanner			:= '';*)
		END_IF
	END_IF
END_FOR

iConfirmFL := 1;
bConfirmReadyFlag := TRUE;

IF bBarcodeTracerInvalidFlag THEN
bConfirmReadyFlag := FALSE;
END_IF

FOR iConfirmFL := 1 TO 10 DO
	IF iConfirmFL >= 1 AND iConfirmFL <= 10 THEN
		IF ARbBarcodeStorageEnable[iConfirmFL] AND ARsHMIBarcodeData_ScanIn[iConfirmFL] = '' THEN
		bConfirmReadyFlag := FALSE;
		END_IF
	END_IF
END_FOR


IF bConfirmPBRE.Q AND bConfirmReadyFlag THEN
ARsBarcodeData_LdBasketInfo 	:= ARsHMIBarcodeData_ScanIn;
ARsHMIBarcodeData_ScanIn 	:= ARsHMIBarcodeData_Empty ;
END_IF


IF NOT bEN THEN
ARsHMIBarcodeData_ScanIn 	:= ARsHMIBarcodeData_Empty ;
END_IF

END_FUNCTION_BLOCK

// ---- FBs/B_JKS_NewFB_V2/FBP-BasketInfoRelated/fbV2_BasketInfoManager.TcPOU
FUNCTION_BLOCK fbV2_BasketInfoManager
VAR_INPUT
	iRecipeChangeFlagDelayTime_Sec : REAL;
END_VAR
VAR_OUTPUT
	bRecipeChangedFlag : BOOL;
	bMinMaxEffChangeFlag : BOOL;

END_VAR
VAR_IN_OUT
	DSV2BasketInfo : DSV2_BasketInfo;
END_VAR

VAR
	tRecipeChangeFlagDelayOffTimer: TON;
	DSV2BasketInfoEmpty : DSV2_BasketInfo;

	iPRNBuffer: INT;
	tMinMaxEffChangeDelayOffTimer: TON;
	iFL: INT;
END_VAR

VAR PERSISTENT
	iPreviousProductRecipeNo: INT;
	ARiCurrentData : ARRAY [1..20] OF INT;
	ARiPreviousData : ARRAY [1..20] OF INT;

END_VAR

(*bMinMaxEffChangeFlag Control*)
ARiCurrentData[1] := DSV2BasketInfo.iCurrentStationNo;
ARiCurrentData[2] := DSV2BasketInfo.iPreviousStationNo;
ARiCurrentData[3] := DSV2BasketInfo.iProductRecipeStepNo;
ARiCurrentData[4] := DSV2BasketInfo.iStationSeqenceRecipeNo;
ARiCurrentData[5] := 0;

ARiCurrentData[6] := DSV2BasketInfo.DSV2MinMaxEffTime.ARiEffTime[1];
ARiCurrentData[7] := DSV2BasketInfo.DSV2MinMaxEffTime.ARiMaxTime[1];
ARiCurrentData[8] := DSV2BasketInfo.DSV2MinMaxEffTime.ARiMinTime[1];
ARiCurrentData[9] := DSV2BasketInfo.DSV2MinMaxEffTime.ARiStnSeqRepNo[1];
ARiCurrentData[10] := DSV2BasketInfo.DSV2MinMaxEffTime.ARiTransferStationNo[1];

ARiCurrentData[11] := DSV2BasketInfo.DSV2MinMaxEffTime.ARiEffTime[2];
ARiCurrentData[12] := DSV2BasketInfo.DSV2MinMaxEffTime.ARiMaxTime[2];
ARiCurrentData[13] := DSV2BasketInfo.DSV2MinMaxEffTime.ARiMinTime[2];
ARiCurrentData[14] := DSV2BasketInfo.DSV2MinMaxEffTime.ARiStnSeqRepNo[2];
ARiCurrentData[15] := DSV2BasketInfo.DSV2MinMaxEffTime.ARiTransferStationNo[2];

ARiCurrentData[16] := DSV2BasketInfo.DSV2MinMaxEffTime.ARiEffTime[3];
ARiCurrentData[17] := DSV2BasketInfo.DSV2MinMaxEffTime.ARiMaxTime[3];
ARiCurrentData[18] := DSV2BasketInfo.DSV2MinMaxEffTime.ARiMinTime[3];
ARiCurrentData[19] := DSV2BasketInfo.DSV2MinMaxEffTime.ARiStnSeqRepNo[3];
ARiCurrentData[20] := DSV2BasketInfo.DSV2MinMaxEffTime.ARiTransferStationNo[3];



iFL := 1;
	FOR iFL := 1 TO 20 DO
		IF iFL > 0 AND iFL <= 20 THEN
			IF ARiCurrentData[iFL] <> ARiPreviousData[iFL] THEN
			bMinMaxEffChangeFlag := TRUE;
			ARiPreviousData[iFL] := ARiCurrentData[iFL];
			END_IF
		END_IF
	END_FOR

IF DSV2BasketInfo.iProductRecipeNo <= 0 THEN
bMinMaxEffChangeFlag := FALSE;
END_IF

tMinMaxEffChangeDelayOffTimer(IN:=bMinMaxEffChangeFlag , PT:=REAL_TO_TIME(iRecipeChangeFlagDelayTime_Sec*1000) , Q=> , ET=> );

IF tMinMaxEffChangeDelayOffTimer.Q THEN
bMinMaxEffChangeFlag := FALSE;
END_IF



(*bRecipeChangedFlag Control*)
tRecipeChangeFlagDelayOffTimer(IN:=bRecipeChangedFlag , PT:=REAL_TO_TIME(iRecipeChangeFlagDelayTime_Sec*1000) , Q=> , ET=> );

	IF tRecipeChangeFlagDelayOffTimer.Q THEN
	bRecipeChangedFlag := FALSE;
	END_IF


	IF DSV2BasketInfo.iProductRecipeNo <> iPreviousProductRecipeNo AND DSV2BasketInfo.iProductRecipeNo > 0 AND DSV2BasketInfo.iProductRecipeNo <= iProductRecipeArrayQty  THEN
	bRecipeChangedFlag := TRUE;
	END_IF

	IF DSV2BasketInfo.iProductRecipeNo <> iPreviousProductRecipeNo THEN
	iPRNBuffer := DSV2BasketInfo.iProductRecipeNo;

		IF NOT bMinMaxEffChangeFlag THEN
			DSV2BasketInfo := DSV2BasketInfoEmpty;
		END_IF

	DSV2BasketInfo.iProductRecipeNo := iPRNBuffer;
	iPRNBuffer := 0;

	iPreviousProductRecipeNo := DSV2BasketInfo.iProductRecipeNo;
	END_IF



(*ProductRecipeNo Move and Availibility Control*)
DSV2BasketInfo.DSV2MinMaxEffTime.iProductRecipeNo := DSV2BasketInfo.iProductRecipeNo;

IF DSV2BasketInfo.iProductRecipeNo > 0 AND DSV2BasketInfo.iProductRecipeNo <= iProductRecipeArrayQty THEN
DSV2BasketInfo.bAvailibility := TRUE;
ELSE
DSV2BasketInfo.bAvailibility := FALSE;
END_IF

END_FUNCTION_BLOCK

// ---- FBs/B_JKS_NewFB/FBP-MachineOperationTimeCounter/fbVacuumPumpTimeCounter.TcPOU
FUNCTION_BLOCK fbVacuumPumpTimeCounter
VAR_INPUT

	bEnable		: BOOL;
	bReset		: BOOL;
	di1stLimitVacPumpTimerSet : DINT;
	di2ndLimitVacPumpTimerSet : DINT;

END_VAR
VAR_OUTPUT

	sTotalTimePV	: STRING;
	b1stLimitVacPumpReachedAlarm: BOOL;
	b2ndLimitVacPumpReachedAlarm: BOOL;

END_VAR
VAR

	TON1			: TON;
	TON2			: TON;
	FBTRIG			: R_TRIG;
	FB1TRIG		: R_TRIG;
	step				: INT;

	Second			: DINT;

END_VAR
VAR PERSISTENT
	Counter				: DINT;
	Minute				: DINT;
	Hour				: DINT;
	Day					: DINT;
END_VAR

TON1(IN:=(bEnable AND NOT TON2.Q) , PT:=T#0.5S , Q=> , ET=> );
TON2(IN:=TON1.Q , PT:=T#0.5S , Q=> , ET=> );
FB1TRIG(CLK:=bReset , Q=> );

IF bEnable THEN
	FBTRIG(CLK:=TON2.Q , Q=> );
END_IF

IF FB1TRIG.Q THEN
	Counter		:= 0;
	Second		:= 0;
	Minute		:= 0;
	Hour		:= 0;
	Day			:= 0;
END_IF

IF bEnable AND FBTRIG.Q THEN
	Second := Second + 1;
END_IF

IF bEnable AND Second >= 60 THEN
	Minute := MInute + 1;
	Second := 0;
END_IF

IF bEnable AND Minute >= 60 THEN
	Hour := hour + 1;
	Minute := 0;
END_IF

IF bEnable AND Hour >= di1stLimitVacPumpTimerSet THEN
	b1stLimitVacPumpReachedAlarm := TRUE;
ELSE
	b1stLimitVacPumpReachedAlarm := FALSE;
END_IF

IF bEnable AND Hour >= di2ndLimitVacPumpTimerSet THEN
	b2ndLimitVacPumpReachedAlarm := TRUE;
ELSE
	b2ndLimitVacPumpReachedAlarm := FALSE;
END_IF

(*
IF bEnable AND Hour >= 24 THEN
	Day := Day +1;
	Hour := 0;
END_IF
*)

sTotalTimePV := CONCAT(DINT_TO_STRING(Day),':');

IF Hour < 10 THEN
sTotalTimePV :=CONCAT(sTotalTimePV,'0');
sTotalTimePV :=CONCAT(sTotalTimePV,DINT_TO_STRING(Hour));
ELSE
sTotalTimePV :=CONCAT(sTotalTimePV,DINT_TO_STRING(Hour));
END_IF

sTotalTimePV := CONCAT(sTotalTimePV,':');

IF Minute < 10 THEN
sTotalTimePV :=CONCAT(sTotalTimePV,'0');
sTotalTimePV :=CONCAT(sTotalTimePV,DINT_TO_STRING(Minute));
ELSE
sTotalTimePV :=CONCAT(sTotalTimePV,DINT_TO_STRING(Minute));
END_IF

sTotalTimePV := CONCAT(sTotalTimePV,':');

IF Second < 10 THEN
sTotalTimePV := CONCAT(sTotalTimePV,'0');
sTotalTimePV := CONCAT(sTotalTimePV,DINT_TO_STRING(Second));
ELSE
sTotalTimePV := CONCAT(sTotalTimePV,DINT_TO_STRING(Second));
END_IF

(***************************************************************)
(*
IF bEnable AND Hour >= 24 THEN
	Day := Day +1;
	Hour := 0;
END_IF

sTotalTimePV := CONCAT(DINT_TO_STRING(Day),':');

IF Hour < 10 THEN
sTotalTimePV :=CONCAT(sTotalTimePV,'0');
sTotalTimePV :=CONCAT(sTotalTimePV,DINT_TO_STRING(Hour));
ELSE
sTotalTimePV :=CONCAT(sTotalTimePV,DINT_TO_STRING(Hour));
END_IF

sTotalTimePV := CONCAT(sTotalTimePV,':');

IF Minute < 10 THEN
sTotalTimePV :=CONCAT(sTotalTimePV,'0');
sTotalTimePV :=CONCAT(sTotalTimePV,DINT_TO_STRING(Minute));
ELSE
sTotalTimePV :=CONCAT(sTotalTimePV,DINT_TO_STRING(Minute));
END_IF

sTotalTimePV := CONCAT(sTotalTimePV,':');

IF Second < 10 THEN
sTotalTimePV := CONCAT(sTotalTimePV,'0');
sTotalTimePV := CONCAT(sTotalTimePV,DINT_TO_STRING(Second));
ELSE
sTotalTimePV := CONCAT(sTotalTimePV,DINT_TO_STRING(Second));
END_IF
*)

END_FUNCTION_BLOCK

// ---- FBs/B_JKS_NewFB_V3/Event/FB3_EventModule.TcPOU
FUNCTION_BLOCK FB3_EventModule 
VAR_INPUT



	bEN								: BOOL;
	bEventRstPBPhysicalInput		: BOOL; // Mapped with Physical Event Reset Push Button Input signal
	bBuzzerRstPBPhysicalInput		: BOOL; // Mapped with Physical Buzzer Reset Push Button Input signal
	bAcknowdgePBPhysicalInput		: BOOL; // Mapped with Physical Acknowledge Push Button Input signal
	bEventRstPB						: REFERENCE TO BOOL; // Mapped with Global variable (Lib-General) with the same name
	bBuzzerRstPB					: REFERENCE TO BOOL; // Mapped with Global variable (Lib-General) with the same name
	bAcknowledgePB					: REFERENCE TO BOOL; // Mapped with Global variable (Lib-General) with the same name
	bAcknowledgeEnable				: BOOL; // TRUE if the EVENT Acknowledge Action will take place (by USER)
	bPowerUpDelayFlag				: BOOL;
	eHmiLanguage					: E_HmiLanguage; (*English:=1, Mandarin:=2, German:=3, French:=4, Portuguese:=5*)
	bActiveEventDisplay_ScrollUp	: BOOL;
	bActiveEventDisplay_ScrollDown	: BOOL;
	bHistoryEventDisplay_ScrollUp	: BOOL;
	bHistoryEventDisplay_ScrollDown	: BOOL;
	
	sCurrentDateAndTimeUser24hr		: STRING(50);

END_VAR
VAR_IN_OUT

END_VAR
VAR_OUTPUT
	bCautionEventOccuredFlag 	: BOOL;
	bWarningEventOccuredFlag 	: BOOL;
	bErrorEventOccuredFlag 		: BOOL;
	iActiveCautionEventCount	: INT;
	iActiveWarningEventCount 	: INT;
	iActiveErrorEventCount	 	: int;
	bBuzzerOutput				: BOOL;
END_VAR
VAR

	bStart								: BOOL; // After Power Up Delay
	bENRE								: R_TRIG;
	bAcknowledgeRE						: R_TRIG;
	iMFL								: INT;
	iFL									: INT;
	iSFL								: INT;
	ARbVirtualEventInputSignal			: ARRAY [1..C_iEventQty] OF BOOL;
	ARbEventOutputRE					: ARRAY [1..C_iEventQty] OF R_TRIG;
	ARbEventOutputFE					: ARRAY [1..C_iEventQty] OF F_TRIG;
	iActiveEventDisplayScrollShiftID 	: INT;
	iHistoryEventDisplayScrollShiftID	: INT;

	bActiveEventDisplay_ScrollUpRE 		: R_TRIG;
	bActiveEventDisplay_ScrollDownRE 	: R_TRIG;
	bActiveScrollIntervalTimerRE		: R_TRIG;
	tmActiveScrollRepeatTimer			: TON;
	tmActiveScrollIntervalTimer			: TON;
	iActiveScrollDelayTime				: INT;

	bHistoryEventDisplay_ScrollUpRE 	: R_TRIG;
	bHistoryEventDisplay_ScrollDownRE 	: R_TRIG;
	bHistoryScrollIntervalTimerRE		: R_TRIG;
	tmHistoryScrollRepeatTimer			: TON;
	tmHistoryScrollIntervalTimer		: TON;
	iHistoryScrollDelayTime				: INT;

	eHmiLanguagePrevious				: E_HmiLanguage;
	
	bEventRstPBPhysicalInputRE			: R_TRIG;
	bBuzzerRstPBPhysicalInputRE			: R_TRIG;
	bAcknowdgePBPhysicalInputRE			: R_TRIG;

	bEventRstPBPhysicalInputFE			: F_TRIG;
	bBuzzerRstPBPhysicalInputFE			: F_TRIG;
	bAcknowdgePBPhysicalInputFE			: F_TRIG;

	bEventRstPBFE						: F_TRIG;
	bBuzzerRstPBFE						: F_TRIG;
	bAcknowdgePBFE						: F_TRIG;	
//	bBool: ARRAY [1..10] OF BOOL;
	
	bStartRE							: R_TRIG;
END_VAR

// Generate RisingEdge
bENRE				(CLK	:= bEN AND (2000 < TO_INT(DSLocalSystemTimeML.sYear)) 	, Q=> );
bAcknowledgeRE		(CLK	:= bAcknowledgePB 										, Q=> );
bStartRE			(CLK	:= bStart 												, Q=> ); // Add by ckk

	// Update HMI Display if the language changed
	IF eHmiLanguagePrevious <> eHmiLanguage THEN

		// Keep current language selection
		eHmiLanguagePrevious := eHmiLanguage;		


		// Language changed detected -> Both Active and History Display need to be update as well	
		mtActiveEventDisplayUpdate(iActiveEventDisplayScrollShiftID);
		mtHistoryEventDisplayUpdate(iHistoryEventDisplayScrollShiftID);


	END_IF

 
	// Trigger Power Up Delay
	IF bEN AND NOT bStart THEN

		IF bPowerUpDelayFlag THEN
			bStart := TRUE;
		END_IF

	ELSIF NOT bEN THEN
		bStart := FALSE;
	END_IF
	
(*	IF bStartRE.Q THEN
		acCaptureEventType();						(* ACTION *)	
	END_IF
*)	
	// Initialised the Active Event State by clearing all event before scanning start & Capture Event Type from AR2dsEventDescriptionCausedRemedy to ARdsEvent
	IF bENRE.Q THEN
		acEventControl_Initialised();				(* ACTION *)
		acCaptureEventType();						(* ACTION *)	
		acEventHistoryRecoveredTimeInitialised();	(* ACTION *)
	END_IF
	
	// Event Scanning Started ***Non-Stop as long as the FB is operating***
	IF bStart THEN
		acEventControl_Scanning();					(* ACTION *)
		acBuzzerOutputControl();					(* ACTION *)
		acPhysicalInputSignalCtrl();				(* ACTION *)		
	END_IF
		

	IF bStart THEN

		// Active Scroll ID Control - To utilised in Active Event Display
		bActiveEventDisplay_ScrollUpRE		(CLK := bActiveEventDisplay_ScrollUp);
		bActiveEventDisplay_ScrollDownRE	(CLK := bActiveEventDisplay_ScrollDown);
		IF bActiveEventDisplay_ScrollUp OR bActiveEventDisplay_ScrollDown THEN
			acActiveScrollShiftIDControl();			(* ACTION *)
		ELSE
			// Reset Scroll delay to default value
			iActiveScrollDelayTime := 1000;
		END_IF


		// History Scroll ID Control - To utilised in History Event Display
		bHistoryEventDisplay_ScrollUpRE		(CLK := bHistoryEventDisplay_ScrollUp);
		bHistoryEventDisplay_ScrollDownRE	(CLK := bHistoryEventDisplay_ScrollDown);
		IF bHistoryEventDisplay_ScrollUp OR bHistoryEventDisplay_ScrollDown THEN
			acHistoryScrollShiftIDControl();		(* ACTION *)
		ELSE
			// Reset Scroll delay to default value
			iHistoryScrollDelayTime := 1000;
		END_IF

		
		IF bBuzzerRstPB THEN
			mtBuzzerReset();
		END_IF
		
		IF bEventRstPB THEN
			mtEventReset();
		END_IF
		
		IF bAcknowledgeEnable AND bAcknowledgeRE.Q THEN
			mtHistoryEventLoggedAcknowledgedTime();
		END_IF
		
		
		
	END_IF

ACTION acActiveScrollShiftIDControl:

		tmActiveScrollRepeatTimer				(IN  := bActiveEventDisplay_ScrollUp OR bActiveEventDisplay_ScrollDown, PT:=T#2S);
		tmActiveScrollIntervalTimer				(IN  := tmActiveScrollRepeatTimer.Q AND NOT tmActiveScrollIntervalTimer.Q, PT:=TO_TIME(iActiveScrollDelayTime));
		bActiveScrollIntervalTimerRE			(CLK := tmActiveScrollIntervalTimer.Q);
		
			// Managed Scroll Delay Time (Long press to reduce the delay time so that the scrolling will speed up
			IF (bActiveEventDisplay_ScrollUp OR bActiveEventDisplay_ScrollDown) AND bActiveScrollIntervalTimerRE.Q THEN
					IF iActiveScrollDelayTime > 100 THEN	
						iActiveScrollDelayTime := iActiveScrollDelayTime - 100;
					END_IF			
			END_IF
			
			IF bActiveEventDisplay_ScrollUp AND NOT bActiveEventDisplay_ScrollDown THEN
		
				// Scroll ID - Up Action
				IF bActiveEventDisplay_ScrollUpRE.Q OR bActiveScrollIntervalTimerRE.Q THEN
					IF iActiveEventDisplayScrollShiftID >= 1 THEN
						iActiveEventDisplayScrollShiftID := iActiveEventDisplayScrollShiftID -1;	// Value can go to lowest "0"
		
						// Update Display	
						mtActiveEventDisplayUpdate(iActiveEventDisplayScrollShiftID);
		
					END_IF
				END_IF
				
			ELSIF NOT bActiveEventDisplay_ScrollUp AND bActiveEventDisplay_ScrollDown THEN	
		
				// Scroll ID - Down Action
				IF bActiveEventDisplay_ScrollDownRE.Q OR bActiveScrollIntervalTimerRE.Q THEN
					IF (iActiveEventDisplayScrollShiftID + C_iEventActiveDisplayQty) < C_iEventActiveLogQty THEN // To ensure Scroll to the lowest display section and not exceed the LogQty
						iActiveEventDisplayScrollShiftID := iActiveEventDisplayScrollShiftID +1;
		
						// Update Display	
						mtActiveEventDisplayUpdate(iActiveEventDisplayScrollShiftID);
		
					END_IF
				END_IF
		
		
			END_IF
END_ACTION

ACTION acBuzzerOutputControl:
		// Buzzer Control - Trigger Buzzer Output

		bBuzzerOutput := FALSE;

		iFL := 1;
		
			FOR iFL := 1 TO C_iEventQty DO
		
		
				IF ARdsEventCtrl[iFL].bEventOutput AND NOT ARdsEventCtrl[iFL].bEventBuzzerStop THEN
					bBuzzerOutput := TRUE;
					iFL := C_iEventQty +1;
				END_IF
		
			END_FOR
END_ACTION

ACTION acCaptureEventType:



// if sEventType is empty or non-recognised wording, it will automatically label it as "ERROR" event type
iFL := 1;

	FOR iFL := 1 TO C_iEventQty DO

		IF AR2dsEventDescriptionCausedRemedy[1][iFL].sEventType = 'Error' THEN 
			ARdsEventCtrl[iFL].eEventType := 2;
		ELSIF AR2dsEventDescriptionCausedRemedy[1][iFL].sEventType = 'Warning' THEN 
			ARdsEventCtrl[iFL].eEventType := 1;
		ELSIF AR2dsEventDescriptionCausedRemedy[1][iFL].sEventType = 'Caution' THEN 
			ARdsEventCtrl[iFL].eEventType := 0;
		ELSE
			ARdsEventCtrl[iFL].eEventType := 2;			
		END_IF
		
	END_FOR
END_ACTION

ACTION acEventControl_Initialised:


iFL := 1;
		
	FOR iFL := 1 TO C_iEventQty DO
		ARdsEventCtrl[iFL].bEventOutput		:= FALSE;
		ARdsEventCtrl[iFL].iDelayTimeEV		:= 0;
		ARdsEventCtrl[iFL].bEventBuzzerStop	:= FALSE;		
	END_FOR
END_ACTION

ACTION acEventControl_Scanning:
// Reset to get ready for status update
	bCautionEventOccuredFlag 	:= FALSE;
	bWarningEventOccuredFlag 	:= FALSE;
	bErrorEventOccuredFlag 		:= FALSE;
	iActiveCautionEventCount	:= 0;
	iActiveWarningEventCount 	:= 0;
	iActiveErrorEventCount	 	:= 0;



// Event Controlling - signal react as output after timer count up
iMFL := 1;

	FOR iMFL := 1 TO C_iEventQty DO

		// To generate Virtual Input follow condition
		IF (ARdsEventCtrl[iMFL].bTest_InvertedInputEn AND NOT ARdsEventCtrl[iMFL].bSignalInput)  
		OR (NOT ARdsEventCtrl[iMFL].bTest_InvertedInputEn AND ARdsEventCtrl[iMFL].bSignalInput) THEN 
			ARbVirtualEventInputSignal[iMFL] := TRUE;	
		ELSE
			ARbVirtualEventInputSignal[iMFL] := FALSE;				
		END_IF
		
		// Action via Virtual Input
		IF ARbVirtualEventInputSignal[iMFL] THEN

			IF (ARdsEventCtrl[iMFL].iDelayTimeSV > ARdsEventCtrl[iMFL].iDelayTimeEV) AND bClockPulse_1Sec THEN
				ARdsEventCtrl[iMFL].iDelayTimeEV := ARdsEventCtrl[iMFL].iDelayTimeEV +1;
			ELSIF (ARdsEventCtrl[iMFL].iDelayTimeSV <= ARdsEventCtrl[iMFL].iDelayTimeEV) THEN
				ARdsEventCtrl[iMFL].bEventOutput := TRUE;
			END_IF

		ELSIF NOT ARbVirtualEventInputSignal[iMFL] THEN

			IF ARdsEventCtrl[iMFL].bHoldingDisable THEN
				ARdsEventCtrl[iMFL].bEventOutput 		:= FALSE;
				ARdsEventCtrl[iMFL].bEventBuzzerStop 	:= FALSE;
			END_IF

				ARdsEventCtrl[iMFL].iDelayTimeEV		:= 0;
	
		END_IF

		// Generate RisingEdge and FailingEdge for every bEventOutput
		ARbEventOutputRE[iMFL](CLK:=ARdsEventCtrl[iMFL].bEventOutput , Q=> );	
		ARbEventOutputFE[iMFL](CLK:=ARdsEventCtrl[iMFL].bEventOutput , Q=> );	

		// RisingEdge Triggered -> Event Occurred -> Event Log
		IF ARbEventOutputRE[iMFL].Q THEN
			mtActiveEventToLogWithOccurredTime(iEventID_ToLog := iMFL);
 			mtHistoryEventToLogWithOccurredTime(iEventID_ToLog := iMFL);

		END_IF
	
		// FallingEdge Triggered -> Event Recovered -> Event Log
		IF ARbEventOutputFE[iMFL].Q THEN
			mtActiveEventRecovered(iEventID_ToClear := iMFL);
 			mtHistoryEventLoggedRecoveredTime(iEventID_ToLog := iMFL);

		END_IF

		// Event Occurred Flag and Count
		IF ARdsEventCtrl[iMFL].bEventOutput THEN
			IF ARdsEventCtrl[iMFL].eEventType = 0 THEN
				bCautionEventOccuredFlag := TRUE;
				iActiveCautionEventCount := iActiveCautionEventCount +1;
			ELSIF ARdsEventCtrl[iMFL].eEventType = 1 THEN
				bWarningEventOccuredFlag := TRUE;
				iActiveWarningEventCount := iActiveWarningEventCount +1;
			ELSIF ARdsEventCtrl[iMFL].eEventType = 2 THEN
				bErrorEventOccuredFlag := TRUE;
				iActiveErrorEventCount := iActiveErrorEventCount +1;
			END_IF
	
		END_IF
		
		// Activate bEventBuzzerStop for "Caution" Event Type Only
		IF ARdsEventCtrl[iMFL].eEventType = 0 THEN
				ARdsEventCtrl[iMFL].bEventBuzzerStop := TRUE;				
		END_IF
	
	END_FOR
END_ACTION

ACTION acEventHistoryRecoveredTimeInitialised:

		iFL := 1;

			// Log Event Recovered Time	to ARdsEventHistoryLog	
			FOR iFL := 1 TO C_iEventHistoryLogQty DO

				IF ARdsEventHistoryLog[iFL].iEventID <> 0 AND ARdsEventHistoryLog[iFL].sTimeAndDate_Recovered = '' THEN								
					ARdsEventHistoryLog[iFL].sTimeAndDate_Recovered												:= sCurrentDateAndTimeUser24hr;

					// If Acknowledge is not Enable, the Acknowledged time will captured follow Recovered time
					IF NOT bAcknowledgeEnable THEN
						ARdsEventHistoryLog[iFL].sTimeAndDate_Acknowledged										:= sCurrentDateAndTimeUser24hr;
					END_IF
				
					// Event Log to MRB (Memory Ring Buffer)				
					FNbCsvEventLogToBuffer(	dsEventHistoryToLog		:= ARdsEventHistoryLog[iFL],
											sDateToLogFIlename		:= DSLocalSystemTimeML.sCurrentDate_General, 
											eCsvActionType			:= eCsvLogData_EventLog, 
											udiCsvMRBCount			=> udiCsvMRBCount, 
											udiCsvMRBUsagePercent	=> udiCsvMRBUsagePercent, 
											bError					=> );

				END_IF

			END_FOR

		
(*
		// After Acknowledged info update -> Display need to be update as well	
		mtHistoryEventDisplayUpdate(iHistoryEventDisplayScrollShiftID);
*)
END_ACTION

ACTION acHistoryScrollShiftIDControl:

		tmHistoryScrollRepeatTimer			(IN  := bHistoryEventDisplay_ScrollUp OR bHistoryEventDisplay_ScrollDown, PT:=T#2S);
		tmHistoryScrollIntervalTimer		(IN  := tmHistoryScrollRepeatTimer.Q AND NOT tmHistoryScrollIntervalTimer.Q, PT:=TO_TIME(iHistoryScrollDelayTime));
		bHistoryScrollIntervalTimerRE		(CLK := tmHistoryScrollIntervalTimer.Q);
		
			// Managed Scroll Delay Time (Long press to reduce the delay time so that the scrolling will speed up
			IF (bHistoryEventDisplay_ScrollUp OR bHistoryEventDisplay_ScrollDown) AND bHistoryScrollIntervalTimerRE.Q THEN
					IF iHistoryScrollDelayTime > 100 THEN	
						iHistoryScrollDelayTime := iHistoryScrollDelayTime - 100;
					END_IF			
			END_IF
			
			IF bHistoryEventDisplay_ScrollUp AND NOT bHistoryEventDisplay_ScrollDown THEN
		
				// Scroll ID - Up Action
				IF bHistoryEventDisplay_ScrollUpRE.Q OR bHistoryScrollIntervalTimerRE.Q THEN
					IF iHistoryEventDisplayScrollShiftID >= 1 THEN
						iHistoryEventDisplayScrollShiftID := iHistoryEventDisplayScrollShiftID -1;	// Value can go to lowest "0"
		
						// Update Display	
						mtHistoryEventDisplayUpdate(iHistoryEventDisplayScrollShiftID);
		
					END_IF
				END_IF
				
			ELSIF NOT bHistoryEventDisplay_ScrollUp AND bHistoryEventDisplay_ScrollDown THEN	
		
				// Scroll ID - Down Action
				IF bHistoryEventDisplay_ScrollDownRE.Q OR bHistoryScrollIntervalTimerRE.Q THEN
					IF (iHistoryEventDisplayScrollShiftID + C_iEventHistoryDisplayQty) < C_iEventHistoryLogQty THEN // To ensure Scroll to the lowest display section and not exceed the LogQty
						iHistoryEventDisplayScrollShiftID := iHistoryEventDisplayScrollShiftID +1;
		
						// Update Display	
						mtHistoryEventDisplayUpdate(iHistoryEventDisplayScrollShiftID);
		
					END_IF
				END_IF
		
		
			END_IF
END_ACTION

ACTION acPhysicalInputSignalCtrl:

// R_TRIG and F_TRIG	
	bEventRstPBPhysicalInputRE	(CLK:=bEventRstPBPhysicalInput 	, Q=> );
	bBuzzerRstPBPhysicalInputRE	(CLK:=bBuzzerRstPBPhysicalInput , Q=> );
	bAcknowdgePBPhysicalInputRE	(CLK:=bAcknowdgePBPhysicalInput , Q=> );
	
	bEventRstPBPhysicalInputFE	(CLK:=bEventRstPBPhysicalInput 	, Q=> );
	bBuzzerRstPBPhysicalInputFE	(CLK:=bBuzzerRstPBPhysicalInput , Q=> );
	bAcknowdgePBPhysicalInputFE	(CLK:=bAcknowdgePBPhysicalInput , Q=> );
	
	bEventRstPBFE				(CLK:=bEventRstPB 				, Q=> );
	bBuzzerRstPBFE				(CLK:=bBuzzerRstPB 				, Q=> );
	bAcknowdgePBFE				(CLK:=bAcknowledgePB 			, Q=> );

	
// EventRstPB
	IF bEventRstPBPhysicalInputRE.Q
	OR bEventRstPBFE.Q AND bEventRstPBPhysicalInput THEN
		bEventRstPB := TRUE;
	END_IF

	IF bEventRstPBPhysicalInputFE.Q THEN
		bEventRstPB := FALSE;
	END_IF
	
// BuzzerRstPB
	IF bBuzzerRstPBPhysicalInputRE.Q
	OR bBuzzerRstPBFE.Q AND bBuzzerRstPBPhysicalInput THEN
		bBuzzerRstPB := TRUE;
	END_IF

	IF bBuzzerRstPBPhysicalInputFE.Q THEN
		bBuzzerRstPB := FALSE;
	END_IF
	
// AcknowledgePB
	IF bAcknowdgePBPhysicalInputRE.Q
	OR bAcknowdgePBFE.Q AND bAcknowdgePBPhysicalInput THEN
		bAcknowledgePB := TRUE;
	END_IF

	IF bAcknowdgePBPhysicalInputFE.Q THEN
		bAcknowledgePB := FALSE;
	END_IF
END_ACTION

METHOD PRIVATE mtActiveEventDisplayUpdate
VAR_INPUT
	iActiveEventDisplayShiftID 	: INT;
END_VAR

VAR
	iCurrentEventID				: INT;
	iFL 						: INT;
END_VAR

		iFL := 1;


			FOR iFL := 1 TO C_iEventActiveDisplayQty DO 
				
				// Create Temporary Variable to easy the reference view
				iCurrentEventID												:= ARdsEventActiveLog[iFL+iActiveEventDisplayShiftID].iEventID; 

				IF iCurrentEventID >= 1 AND iCurrentEventID <= C_iEventQty THEN						
					// Generate View/Display				
					ARdsEventActiveDisplay[iFL].iEventID						:= iCurrentEventID;
					ARdsEventActiveDisplay[iFL].sEventCode						:= AR2dsEventDescriptionCausedRemedy[eHmiLanguage][iCurrentEventID].sEventCode;
					ARdsEventActiveDisplay[iFL].sEventType						:= AR2dsEventDescriptionCausedRemedy[eHmiLanguage][iCurrentEventID].sEventType;
					ARdsEventActiveDisplay[iFL].sLocation						:= AR2dsEventDescriptionCausedRemedy[eHmiLanguage][iCurrentEventID].sLocation;
					ARdsEventActiveDisplay[iFL].sSubLocation					:= AR2dsEventDescriptionCausedRemedy[eHmiLanguage][iCurrentEventID].sSubLocation;
					
					ARdsEventActiveDisplay[iFL].sDescription					:= AR2dsEventDescriptionCausedRemedy[eHmiLanguage][iCurrentEventID].sDescription;
					ARdsEventActiveDisplay[iFL].sCaused							:= AR2dsEventDescriptionCausedRemedy[eHmiLanguage][iCurrentEventID].sCaused;
					ARdsEventActiveDisplay[iFL].sRemedy							:= AR2dsEventDescriptionCausedRemedy[eHmiLanguage][iCurrentEventID].sRemedy;
					
					ARdsEventActiveDisplay[iFL].sTimeAndDate_Occurred			:= ARdsEventActiveLog[iFL+iActiveEventDisplayShiftID].sTimeAndDate_Occurred;


				ELSE
					// Load Empty data since the EventID is 0		
					ARdsEventActiveDisplay[iFL] := DSEventActiveDisplayEmpty;
					ARdsEventActiveLog[iFL] := dsEventActiveLogEmpty;
				END_IF
			END_FOR
END_METHOD

METHOD PRIVATE mtActiveEventRecovered
VAR_INPUT
	iEventID_ToClear 	: INT;
END_VAR

VAR
	iFL					: INT;
	iSFL				: INT;
END_VAR
		iFL := 1;

			FOR iFL := 1 TO C_iEventActiveLogQty DO

				IF ARdsEventActiveLog[iFL].iEventID <> 0 THEN			

					IF ARdsEventActiveLog[iFL].iEventID = iEventID_ToClear THEN								
						// Found and Clear the specified Event
						ARdsEventActiveLog[iFL] := DSEventActiveLogEmpty;

						//Shift bottom event to replaced the clear row
						iSFL := 1;	
							FOR iSFL := 1 TO C_iEventActiveLogQty DO
								IF iFL+iSFL <= C_iEventActiveLogQty THEN
									IF ARdsEventActiveLog[iFL+iSFL].iEventID <> 0 THEN
										ARdsEventActiveLog[iFL+iSFL-1] := ARdsEventActiveLog[iFL+iSFL];
									ELSE
										ARdsEventActiveLog[iFL+iSFL-1] := DSEventActiveLogEmpty;
										
									END_IF
								ELSE					
									ARdsEventActiveLog[C_iEventActiveLogQty].iEventID := 0;
									iSFL := C_iEventActiveLogQty +1;									
								END_IF
							END_FOR

						// Found one matched Event ID And Done -> Stop the FL since the Found Event Log has been clear 
						iFL := C_iEventActiveLogQty +1;		

					END_IF

				ELSE
					iFL := C_iEventActiveLogQty +1;
				END_IF
				
			END_FOR

		// After Acknowledged info update -> Display need to be update as well	
			mtActiveEventDisplayUpdate(iActiveEventDisplayScrollShiftID);
END_METHOD

// mtActiveEventToLog TRUE = Complete without Error, mtActiveEventToLog FALSE = Active Log is overflowed 
METHOD PRIVATE mtActiveEventToLogWithOccurredTime : BOOL
VAR_INPUT
	iEventID_ToLog 	: INT;
END_VAR

VAR
	iFL 			: INT;
END_VAR
		// Prepare for completion (if no error, this signal (mtActiveEventToLog) will stay ON
		mtActiveEventToLogWithOccurredTime := TRUE;	

		// Check if overflow on the active log quantity  
		IF ARdsEventActiveLog[C_iEventActiveLogQty].iEventID <> 0 THEN

			// Trigger Error due to overflow in active log quantity
			mtActiveEventToLogWithOccurredTime := FALSE;	

		ELSE


			iFL := 1;

			FOR iFL := 1 TO C_iEventActiveLogQty DO

				IF iFL >= 1 AND iFL < C_iEventActiveLogQty THEN		
					
						// Shift one index to free up [1] to log latest Event
						IF ARdsEventActiveLog[C_iEventActiveLogQty-iFL].iEventID <> 0 THEN			
							ARdsEventActiveLog[C_iEventActiveLogQty-iFL+1] := ARdsEventActiveLog[C_iEventActiveLogQty-iFL];		
						END_IF
	
				END_IF

			END_FOR


			// Log Latest Event and Occurred Time
			IF mtActiveEventToLogWithOccurredTime THEN
				ARdsEventActiveLog[1].iEventID 				:= iEventID_ToLog;				
				ARdsEventActiveLog[1].sTimeAndDate_Occurred	:= sCurrentDateAndTimeUser24hr;
			END_IF
				
			// After Acknowledged info update -> Display need to be update as well	
				mtActiveEventDisplayUpdate(iActiveEventDisplayScrollShiftID);
			
		END_IF
END_METHOD

METHOD PRIVATE mtBuzzerReset

VAR
	iFL				: INT;
END_VAR

		// Buzzer Control - Stop Buzzer Condition

		iFL := 1;
		
			FOR iFL := 1 TO C_iEventQty DO
				
				IF ARdsEventCtrl[iFL].bEventOutput THEN
					IF  (ARdsEventCtrl[iFL].eEventType = 1 OR ARdsEventCtrl[iFL].eEventType = 2) THEN
						ARdsEventCtrl[iFL].bEventBuzzerStop := TRUE;
					END_IF
				END_IF
				
			END_FOR
END_METHOD

METHOD PRIVATE mtEventReset
VAR_INPUT
END_VAR

VAR
	iFL				: INT;
END_VAR

		// Event Reset

		iFL := 1;
		
			FOR iFL := 1 TO C_iEventQty DO
				
				IF NOT ARbVirtualEventInputSignal[iFL] THEN
					ARdsEventCtrl[iFL].bEventOutput 		:= FALSE;
					ARdsEventCtrl[iFL].bEventBuzzerStop 	:= FALSE;
				END_IF
				
			END_FOR
END_METHOD

METHOD PRIVATE mtHistoryEventDisplayUpdate
VAR_INPUT
	iHistoryEventDisplayShiftID 	: INT;
END_VAR

VAR
	iCurrentEventID					: INT;
	iFL								: INT;
END_VAR

		iFL := 1;


			FOR iFL := 1 TO C_iEventHistoryDisplayQty DO 
				
				// Create Temporary Variable to easy the reference view
				iCurrentEventID												:= ARdsEventHistoryLog[iFL+iHistoryEventDisplayShiftID].iEventID; 

				IF iCurrentEventID >= 1 AND iCurrentEventID <= C_iEventQty THEN					
					// Generate View/Display				
					ARdsEventHistoryDisplay[iFL].iEventID						:= iCurrentEventID;
					ARdsEventHistoryDisplay[iFL].sEventCode					:= AR2dsEventDescriptionCausedRemedy[eHmiLanguage][iCurrentEventID].sEventCode;
					ARdsEventHistoryDisplay[iFL].sEventType					:= AR2dsEventDescriptionCausedRemedy[eHmiLanguage][iCurrentEventID].sEventType;
					ARdsEventHistoryDisplay[iFL].sLocation					:= AR2dsEventDescriptionCausedRemedy[eHmiLanguage][iCurrentEventID].sLocation;
					ARdsEventHistoryDisplay[iFL].sSubLocation					:= AR2dsEventDescriptionCausedRemedy[eHmiLanguage][iCurrentEventID].sSubLocation;
					
					ARdsEventHistoryDisplay[iFL].sDescription					:= AR2dsEventDescriptionCausedRemedy[eHmiLanguage][iCurrentEventID].sDescription;
					ARdsEventHistoryDisplay[iFL].sCaused						:= AR2dsEventDescriptionCausedRemedy[eHmiLanguage][iCurrentEventID].sCaused;
					ARdsEventHistoryDisplay[iFL].sRemedy						:= AR2dsEventDescriptionCausedRemedy[eHmiLanguage][iCurrentEventID].sRemedy;
					
					ARdsEventHistoryDisplay[iFL].sTimeAndDate_Occurred		:= ARdsEventHistoryLog[iFL+iHistoryEventDisplayShiftID].sTimeAndDate_Occurred;
					ARdsEventHistoryDisplay[iFL].sTimeAndDate_Acknowledged	:= ARdsEventHistoryLog[iFL+iHistoryEventDisplayShiftID].sTimeAndDate_Acknowledged;
					ARdsEventHistoryDisplay[iFL].sTimeAndDate_Recovered		:= ARdsEventHistoryLog[iFL+iHistoryEventDisplayShiftID].sTimeAndDate_Recovered;

				ELSE
					// Load Empty data since the EventID is 0		
					ARdsEventHistoryDisplay[iFL] := DSEventHistoryDisplayEmpty;
					ARdsEventHistoryLog[iFL] := dsEventHistoryLogEmpty;
				END_IF
			END_FOR
END_METHOD

METHOD PRIVATE mtHistoryEventLoggedAcknowledgedTime
VAR_INPUT
END_VAR

VAR
	iFL				: INT;
END_VAR
		iFL := 1;

			// Log Event Acknowledged Time		
			FOR iFL := 1 TO C_iEventHistoryLogQty DO

				IF ARdsEventHistoryLog[iFL].iEventID <> 0 AND ARdsEventHistoryLog[iFL].sTimeAndDate_Acknowledged = '' THEN								
					ARdsEventHistoryLog[iFL].sTimeAndDate_Acknowledged 	:= sCurrentDateAndTimeUser24hr;
				END_IF

			END_FOR



		// After Acknowledged info update -> Display need to be update as well	
			mtHistoryEventDisplayUpdate(iHistoryEventDisplayScrollShiftID);
END_METHOD

METHOD PRIVATE mtHistoryEventLoggedRecoveredTime
VAR_INPUT
	iEventID_ToLog : INT;
END_VAR

VAR
	iFL				: INT;
END_VAR
		iFL := 1;

			// Log Event Recovered Time	to ARdsEventHistoryLog	
			FOR iFL := 1 TO C_iEventHistoryLogQty DO

				IF ARdsEventHistoryLog[iFL].iEventID = iEventID_ToLog AND ARdsEventHistoryLog[iFL].sTimeAndDate_Recovered = '' THEN								
					ARdsEventHistoryLog[iFL].sTimeAndDate_Recovered												:= sCurrentDateAndTimeUser24hr;

					// If Acknowledge is not Enable, the Acknowledged time will captured follow Recovered time
					IF NOT bAcknowledgeEnable THEN
						ARdsEventHistoryLog[iFL].sTimeAndDate_Acknowledged											:= sCurrentDateAndTimeUser24hr;
					END_IF

					// Event Log to MRB (Memory Ring Buffer)				
					FNbCsvEventLogToBuffer(	dsEventHistoryToLog		:= ARdsEventHistoryLog[iFL],
											sDateToLogFIlename		:= DSLocalSystemTimeML.sCurrentDate_General, 
											eCsvActionType			:= eCsvLogData_EventLog, 
											udiCsvMRBCount			=> udiCsvMRBCount, 
											udiCsvMRBUsagePercent	=> udiCsvMRBUsagePercent, 
											bError					=> );
				
				END_IF


			END_FOR

			

		// After Acknowledged info update -> Display need to be update as well	
			mtHistoryEventDisplayUpdate(iHistoryEventDisplayScrollShiftID);
END_METHOD

METHOD PRIVATE mtHistoryEventToLogWithOccurredTime
VAR_INPUT
	iEventID_ToLog 	: INT;
END_VAR

VAR
	iFL				: INT;
END_VAR
		// Log Event - History Log + Occurred Time Log 
		iFL := 1;

			// Shift one index to free up [1] to log latest Event		
			FOR iFL := 1 TO C_iEventHistoryLogQty DO

				IF iFL >= 1 AND iFL < C_iEventHistoryLogQty THEN								
					ARdsEventHistoryLog[C_iEventHistoryLogQty-iFL+1]			:= ARdsEventHistoryLog[C_iEventHistoryLogQty-iFL];
				END_IF
			END_FOR

		// Log Latest Event and Occurred Time
		ARdsEventHistoryLog[1].iEventID					:= iEventID_ToLog;
		ARdsEventHistoryLog[1].sTimeAndDate_Occurred		:= sCurrentDateAndTimeUser24hr;
		ARdsEventHistoryLog[1].sTimeAndDate_Acknowledged	:= '';
		ARdsEventHistoryLog[1].sTimeAndDate_Recovered		:= '';


		// After Acknowledged info update -> Display need to be update as well	
			mtHistoryEventDisplayUpdate(iHistoryEventDisplayScrollShiftID);
END_METHOD

END_FUNCTION_BLOCK

// ---- FBs/B_JKS_NewFB_V3/CSV/FB3_CsvHandler.TcPOU
FUNCTION_BLOCK FB3_CsvHandler

VAR_INPUT
	bEn 							: BOOL;
	bReset							: BOOL;
	bShutdownRequestFlag 			: BOOL;
	bClearErrorLog					: REFERENCE TO BOOL;
END_VAR

VAR_OUTPUT
	bIdle							: BOOL;
	bProgress						: BOOL;
	bReadyToShutdownFlag 			: BOOL;
	bError							: BOOL;
	bErrorCaseId					: INT;
END_VAR                     		
                            		
VAR_IN_OUT                  		
	udiCsvMRBCount					: UDINT;
	udiCsvMRBUsagePercent 			: UDINT;	
END_VAR
VAR
	dsCsvLog						: DS_CsvLog;
	dsCsvLog_Previous				: DS_CsvLog;
	dsCsvLog_Empty					: DS_CsvLog;
	bScanOnce						: BOOL := TRUE;
	iCase							: INT;
	
	fbFileOpen						: FB_FileOpen;
	fbFilePuts						: FB_FilePuts;
	fbFileSeek						: FB_FileSeek;
	fbFileClose						: FB_FileClose;
	fbFileRename					: FB_FileRename;	
	fbFileDelete					: FB_FileDelete;	
	bFileOpened						: BOOL; // To keep trace if the file opened and havent close
	
	ARbScanOnce						: ARRAY [1..99] OF BOOL;
	ARbScanOnce_Empty				: ARRAY [1..99] OF BOOL;
	iFL								: INT;
	bError_NonImportant				: BOOL;
	iEventLogTitleStep				: INT;
	sEventLogString					: STRING(255);
	bEventLogTitleDone				: BOOL;
	dsEventHistoryDummy 			: DS_EventHistory;
	sDateToLogFilename: STRING;
END_VAR
VAR PERSISTENT
sPreviousEventLogDate : STRING;
END_VAR

	// Detect Next Day and trigger EventLog Filename Generate (from CS_ to CSV)
	IF sPreviousEventLogDate = '' THEN	// Prevent if Persistent currupted and caused the date initialised, this step is to avoid trigger CSV Generate. 
		sPreviousEventLogDate := dsLocalSystemTimeML.sCurrentDate_General;
	END_IF

	IF 	sPreviousEventLogDate <> dsLocalSystemTimeML.sCurrentDate_General THEN
		sDateToLogFilename	:= 	sPreviousEventLogDate;		
		sPreviousEventLogDate := dsLocalSystemTimeML.sCurrentDate_General;
		// Event Log to MRB (Memory Ring Buffer)				
		FNbCsvEventLogToBuffer(	dsEventHistoryToLog		:= dsEventHistoryDummy,
								sDateToLogFIlename		:= sDateToLogFilename, 
								eCsvActionType			:= eCsvGenerate_EventLog, 
								udiCsvMRBCount			=> udiCsvMRBCount, 
								udiCsvMRBUsagePercent	=> udiCsvMRBUsagePercent, 
								bError					=> );			 
	END_IF


	IF bScanOnce THEN
		//readout the current MRBCount and UsagePecentage
		FNbCsvReadWithoutRemoveBuffer(
										dsCsvLog				=>	dsCsvLog , 
										udiCsvMRBCount			=> udiCsvMRBCount, 
										udiCsvMRBUsagePercent	=> udiCsvMRBUsagePercent );	
		bScanOnce := FALSE;	
	END_IF

	
		
	IF bEN  AND NOT bReset THEN
				IF iCase < 1 THEN iCase := 1; END_IF
	ELSE
				iCase					:= 0;
	END_IF
	

	// RESET/Clear CSV Error Log
IF iFL >=1 THEN	
	IF bClearErrorLog THEN
		FOR iFL := 1 TO 100 DO
			ARdsCsvErrorLog[iFL] := dsCsvErrorLog_Empty;
		END_FOR
		bClearErrorLog := FALSE;		
	END_IF
END_IF	
CASE iCase OF
	0: // FunctionBlock Disable
				bIdle 					:= FALSE;
				bProgress 				:= FALSE;	
				bReadyToShutdownFlag 	:= FALSE;
				bError					:= FALSE;
				bErrorCaseId			:= 0;
				dsCsvLog				:=	dsCsvLog_Empty;
				dsCsvLog_Previous		:=	dsCsvLog_Empty;
				ARbScanOnce				:=	ARbScanOnce_Empty;
				bFileOpened				:= FALSE;
				
	1: // Idling

		
		// Indicator Handling
		IF NOT bShutdownRequestFlag THEN
			IF udiCsvMRBCount = 0 THEN
				bIdle 					:= TRUE;
				bProgress 				:= FALSE;	
				bReadyToShutdownFlag 	:= FALSE;
			ELSE
				bIdle 					:= FALSE;
				bProgress 				:= TRUE;	
				bReadyToShutdownFlag 	:= FALSE;
			END_IF
		ELSE
			IF udiCsvMRBCount = 0 THEN
				bIdle 					:= TRUE;
				bProgress 				:= FALSE;	
				bReadyToShutdownFlag 	:= TRUE;
			ELSE
				bIdle 					:= FALSE;
				bProgress 				:= TRUE;	
				bReadyToShutdownFlag 	:= FALSE;
			END_IF
			
		END_IF
 
		IF udiCsvMRBCount <> 0 THEN
				iCase	:= 2;
		END_IF
	
	
	2: // Read Without Remove from MRB (Memory Ring Buffer) 
	
		FNbCsvReadWithoutRemoveBuffer(
							dsCsvLog				=>	dsCsvLog , 
							udiCsvMRBCount			=>	udiCsvMRBCount , 
							udiCsvMRBUsagePercent	=>	udiCsvMRBUsagePercent , 	
							bError					=>	bError );
		
		IF NOT bError THEN
				iCase 			:= 3;
		ELSE
			FNbCsvErrorLog(iCaseId:= iCase, udiErrorId:= 9999, dsCsvLog:= dsCsvLog);
			bErrorCaseId 	:= iCase;
			iCase			:= 97; // Close File and go Case 99 to wait
		END_IF
		
	
	3: // Prepare for Write Process	
		
		CASE dsCsvLog.eLogAction OF

			eCsvLogData_EventLog:
				iCase 				:= 10; // Proceed File Open
				fbFileOpen(nMode	:= FOPEN_MODEREAD OR FOPEN_MODEPLUS OR FOPEN_MODETEXT);
			
			eCsvNewFile_EventLog, eCsvNewFile_CarrierReport, eCsvLogData_CarrierReport:			
				iCase 				:= 10; // Proceed File Open
				fbFileOpen(nMode	:= FOPEN_MODEAPPEND OR FOPEN_MODETEXT);

			eCsvGenerate_CarrierReport, eCsvGenerate_EventLog:
				iCase	:= 30; // Rename CSV File	
				
		END_CASE

	10: // File Open
		
		IF NOT bFileOpened THEN
			fbFileOpen(bExecute	:= FALSE );
			fbFileOpen(
				sPathName		:= CONCAT(dsCsvLog.sPathAndFilename,'.CS_'), 
				ePath			:= PATH_GENERIC, 
				bExecute		:= TRUE );				
		ELSE
				iCase			:= 12; // Proceed FileSeek 
		END_IF
		
		IF fbFileOpen.bBusy THEN
				iCase			:= 11; // FileOpen in progress, go to check point
		END_IF


	11: // File Open - Check point
	
		fbFileOpen(bExecute	:= FALSE );
		IF NOT fbFileOpen.bBusy THEN
			IF NOT fbFileOpen.bError THEN
				iCase			:= 12; // Proceed FileSeek 
				bFileOpened		:= TRUE;
			ELSE
				IF fbFileOpen.nErrId = 1804 AND dsCsvLog.eLogAction = eCsvLogData_EventLog THEN
					iCase				:= 41; // Proceed New File with Title
				ELSE		
					FNbCsvErrorLog(iCaseId:= iCase, udiErrorId:= fbFileOpen.nErrId, dsCsvLog:= dsCsvLog);
					bErrorCaseId 	:= iCase;
					iCase			:= 20; // Proceed Remove MRB, Check & Close File, Clear Current Log in MRB and proceed Next Log
				END_IF
			END_IF				
		END_IF

		
		41: // New file
	
			fbFileOpen(bExecute	:= FALSE );
			fbFileOpen(
				nMode			:= FOPEN_MODEWRITE OR FOPEN_MODEPLUS OR FOPEN_MODETEXT,
				sPathName		:= CONCAT(dsCsvLog.sPathAndFilename,'.CS_'), 
				ePath			:= PATH_GENERIC, 
				bExecute		:= TRUE );				
			
			IF fbFileOpen.bBusy THEN
					iCase		:= 42; // FileOpen in progress, go to check point
			END_IF

		42: // New File Open - Check point
		
			fbFileOpen(bExecute	:= FALSE );
			IF NOT fbFileOpen.bBusy THEN
				IF NOT fbFileOpen.bError THEN
					iCase				:= 43; // Proceed Write Title 
					iEventLogTitleStep	:= 1;
					bEventLogTitleDone	:= FALSE;
					bFileOpened			:= TRUE;
				ELSE
					FNbCsvErrorLog(iCaseId:= iCase, udiErrorId:= fbFileOpen.nErrId, dsCsvLog:= dsCsvLog);
					bErrorCaseId 	:= iCase;
					iCase			:= 20; // Proceed Remove MRB, Check & Close File, Clear Current Log in MRB and proceed Next Log
				END_IF				
			END_IF
	
	
		43: // File Puts (Write Title)
					// Prepare Data
					dsCsvReport.ARsLogTitle_EventLog[1] := 'Occurred Time';
					dsCsvReport.ARsLogTitle_EventLog[2] := 'Acknowledged Time';
					dsCsvReport.ARsLogTitle_EventLog[3] := 'Recovered Time';
					dsCsvReport.ARsLogTitle_EventLog[4] := 'Event ID';
					dsCsvReport.ARsLogTitle_EventLog[5] := 'Event Code';
					dsCsvReport.ARsLogTitle_EventLog[6] := 'Event Type';
					dsCsvReport.ARsLogTitle_EventLog[7] := 'Main Location';
					dsCsvReport.ARsLogTitle_EventLog[8] := 'Sub Location';
					dsCsvReport.ARsLogTitle_EventLog[9] := 'Description';
	//				dsCsvReport.ARsLogTitle_EventLog[10] := ;

					IF dsCsvReport.iNumOfData_LogTitle_EventLog >= iEventLogTitleStep THEN
						sEventLogString := concat(dsCsvReport.ARsLogTitle_EventLog[iEventLogTitleStep],','); 
					ELSE
						sEventLogString := '$N';
						bEventLogTitleDone := TRUE;
					END_IF	
						
						
				fbFilePuts(	bExecute:= FALSE );
				fbFilePuts(	
					hFile			:= fbFileOpen.hFile, 
					sLine			:= sEventLogString, 
					bExecute		:= TRUE );	
	
			IF fbFilePuts.bBusy THEN
					iCase			:= 44; // FilePuts in progress, go to check point	
			END_IF
	
		44: // File Puts - Check point
		
			fbFilePuts(	bExecute:= FALSE );
			IF NOT fbFilePuts.bBusy THEN
				IF NOT fbFilePuts.bError THEN
					IF NOT bEventLogTitleDone THEN
						iCase				:= 43; // Continue Write Event Log Title
						iEventLogTitleStep 	:= iEventLogTitleStep + 1; 
					ELSE
						iCase 				:= 12; // Title Done, Write data
						bEventLogTitleDone	:= FALSE;
					END_IF
					
				ELSE
					FNbCsvErrorLog(iCaseId:= iCase, udiErrorId:= fbFilePuts.nErrId, dsCsvLog:= dsCsvLog);
					bErrorCaseId 	:= iCase;
					iCase			:= 20; // Proceed Remove MRB, Check & Close File, Clear Current Log in MRB and proceed Next Log
				END_IF				
			END_IF

				
	12: // File Seek
	
			fbFileSeek(	bExecute:= FALSE );
			fbFileSeek(	
				eOrigin			:= SEEK_END,
				hFile			:= fbFileOpen.hFile, 
				bExecute		:= TRUE );	
				
		IF fbFileSeek.bBusy THEN
				iCase			:= 13; // FileSeek in progress, go to check point
		END_IF

	13: // File Seek - Check point

		fbFileSeek(	bExecute:= FALSE );
		IF NOT fbFileSeek.bBusy THEN
			IF NOT fbFileSeek.bError THEN
				iCase			:= 14; // Proceed FilePuts (Write data) 
			ELSE
				FNbCsvErrorLog(iCaseId:= iCase, udiErrorId:= fbFileSeek.nErrId, dsCsvLog:= dsCsvLog);
				bErrorCaseId 	:= iCase;
				iCase			:= 20; // Proceed Remove MRB, Check & Close File, Clear Current Log in MRB and proceed Next Log
			END_IF				
		END_IF

	14: // File Puts (Write Data)
			fbFilePuts(	bExecute:= FALSE );
			fbFilePuts(	
				hFile			:= fbFileOpen.hFile, 
				sLine			:= dsCsvLog.sLogString, 
				bExecute		:= TRUE );	

		IF fbFilePuts.bBusy THEN
				iCase			:= 15; // FilePuts in progress, go to check point	
		END_IF

	15: // File Puts - Check point
	
		fbFilePuts(	bExecute:= FALSE );
		IF NOT fbFilePuts.bBusy THEN
			IF NOT fbFilePuts.bError THEN
				iCase			:= 20; // Proceed Remove MRB, Check & Close File, Clear Current Log in MRB and proceed Next Log
			ELSE
				FNbCsvErrorLog(iCaseId:= iCase, udiErrorId:= fbFilePuts.nErrId, dsCsvLog:= dsCsvLog);
				bErrorCaseId 	:= iCase;
				iCase			:= 20; // Proceed Remove MRB, Check & Close File, Clear Current Log in MRB and proceed Next Log
			END_IF				
		END_IF

	20: // Remove MRB and put into dsCsvLog_Previous
	IF NOT ARbScanOnce[20] THEN 	
		FNbCsvReadAndRemoveBuffer(
							dsCsvLog				=>	dsCsvLog_Previous , 
							udiCsvMRBCount			=>	udiCsvMRBCount , 
							udiCsvMRBUsagePercent	=>	udiCsvMRBUsagePercent , 	
							bError					=>	bError );
		ARbScanOnce[20] := TRUE;
	END_IF
		
		IF NOT bError THEN
			IF udiCsvMRBCount >= 1 THEN
				iCase 			:= 21; // Proceed to Check and determine whether to close file or not
				ARbScanOnce[20] := FALSE;
			ELSE
				iCase			:= 22; // Proceed File Close
				ARbScanOnce[20] := FALSE;				
			END_IF
		ELSE
			FNbCsvErrorLog(iCaseId:= iCase, udiErrorId:= 9999, dsCsvLog:= dsCsvLog);
			bErrorCaseId 	:= iCase;
			ARbScanOnce[20] := FALSE;
			iCase			:= 97; // Close File and go Case 99 to wait
		END_IF


	21: // 	Check and determine whether to close file or not		
		
	IF NOT ARbScanOnce[21] THEN 	
		FNbCsvReadWithoutRemoveBuffer(
							dsCsvLog				=>	dsCsvLog , 
							udiCsvMRBCount			=>	udiCsvMRBCount , 
							udiCsvMRBUsagePercent	=>	udiCsvMRBUsagePercent , 	
							bError					=>	bError_NonImportant );
		ARbScanOnce[21] := TRUE;
	END_IF
		
		IF NOT bError_NonImportant THEN	
			IF dsCsvLog_Previous.sPathAndFilename = dsCsvLog.sPathAndFilename AND dsCsvLog_Previous.eLogAction = dsCsvLog.eLogAction AND dsCsvLog.eLogAction <> eCsvGenerate_CarrierReport AND dsCsvLog.eLogAction <> eCsvGenerate_EventLog THEN // Matched, Skipped File Open
				iCase			:= 14; // Proceed FilePuts (Write data) 
				ARbScanOnce[21] := FALSE;
					
			ELSE
				iCase			:= 22; // Proceed File Close
				ARbScanOnce[21] := FALSE;
			END_IF			
		ELSE 
			iCase				:= 22; // Possible the Buffer is empty, so just proceed to File Close 1 
			ARbScanOnce[21]		:= FALSE;
			bError_NonImportant := FALSE;
		END_IF
	
	
	22: // File Close		

			fbFileClose(	bExecute:= FALSE );
			fbFileClose(	
				hFile			:= fbFileOpen.hFile, 
				bExecute		:= TRUE );	

		IF fbFileClose.bBusy THEN
				iCase			:= 23; // FileClose in progress, go to check point
		END_IF


	23: // File Close - Check point
	
		fbFileClose(	bExecute:= FALSE );
		IF NOT fbFileClose.bBusy THEN
			IF NOT fbFileClose.bError THEN
				iCase			:= 1; // Done -> Check next Log or Idle
				bFileOpened		:= FALSE;
			ELSE
				FNbCsvErrorLog(iCaseId:= iCase, udiErrorId:= fbFileClose.nErrId, dsCsvLog:= dsCsvLog);
				bErrorCaseId 	:= iCase;
				iCase			:= 1; // Nothing much can do, just proceed next Log or Idle
			END_IF				
		END_IF
	

	30: // Rename CSV 


	
			fbFileRename(	bExecute:= FALSE );
			fbFileRename(	
					sOldName		:= CONCAT(dsCsvLog.sPathAndFilename,'.CS_'), 
					sNewName		:= CONCAT(dsCsvLog.sPathAndFilename,'.CSV'), 
					ePath			:= PATH_GENERIC,
					bExecute		:= TRUE );

		IF fbFileRename.bBusy THEN
				iCase			:= 31; // RenameCSV in progress, go to check point
		END_IF

	31: // Rename CSV - Check point
	
		fbFileRename(	bExecute:= FALSE );
		IF NOT fbFileRename.bBusy THEN
			IF NOT fbFileRename.bError THEN
				iCase			:= 32; // Done -> Proceed Remove MRB 
			ELSE
				FNbCsvErrorLog(iCaseId:= iCase, udiErrorId:= fbFileRename.nErrId, dsCsvLog:= dsCsvLog);
				bErrorCaseId 	:= iCase;
				iCase			:= 32; // Nothing much can do, just proceed Remove MRB
			END_IF				
		END_IF
	
	32: // Remove MRB and put into dsCsvLog_Previous
		
	IF NOT ARbScanOnce[32] THEN 	
		FNbCsvReadAndRemoveBuffer(
							dsCsvLog				=>	dsCsvLog_Previous , 
							udiCsvMRBCount			=>	udiCsvMRBCount , 
							udiCsvMRBUsagePercent	=>	udiCsvMRBUsagePercent , 	
							bError					=>	bError );
		ARbScanOnce[32] := TRUE;
	END_IF
		
		IF NOT bError THEN
			iCase 			:= 1; // Done -> Check next Log or Idle
			ARbScanOnce[32] := FALSE;
		ELSE
			FNbCsvErrorLog(iCaseId:= iCase, udiErrorId:= 9999, dsCsvLog:= dsCsvLog);
			bErrorCaseId 	:= iCase;
			ARbScanOnce[32] := FALSE;
			iCase			:= 97; // Close File and go Case 99 to wait
		END_IF

	97: // File Close (with Error Reading from Buffer)		

			fbFileClose(	bExecute:= FALSE );
			fbFileClose(	
				hFile			:= fbFileOpen.hFile, 
				bExecute		:= TRUE );	

		IF fbFileClose.bBusy THEN
				iCase			:= 98; // FileClose in progress, go to check point
		END_IF


	98: // File Close - Check point (with Error Reading from Buffer)
	
		fbFileClose(	bExecute:= FALSE );
		IF NOT fbFileClose.bBusy THEN
			IF NOT fbFileClose.bError THEN
					iCase			:= 99;
					bFileOpened		:= FALSE;
			ELSE
				FNbCsvErrorLog(iCaseId:= iCase, udiErrorId:= fbFileClose.nErrId, dsCsvLog:= dsCsvLog);
				bErrorCaseId 	:= iCase;
				iCase			:= 99; 
			END_IF				
		END_IF
	


				
	99:; // Error, Stay here


END_CASE

END_FUNCTION_BLOCK

// ---- FBs/B_JKS_NewFB_V2/FBP-StationRelated/fbV2_MainStationProcess.TcPOU
FUNCTION_BLOCK fbV2_MainStationProcess

(*************************************************************** Ver.B1 - fbV2_StnSeqProcess - 161101 **************************************************************]

 	- Add 'bEffTimePriorityEn' to cutoff the process once effective time reached.																	
	- Change naming from 'bProcessCompleteBasedMasterTime' to 'bMinMaxEn'. 
	- 	
	- 
[****************************************************************************************************************************************************************************************************)

VAR_INPUT
	(*fbStnSeqProcess*)
	bAutoStartPbEn									: BOOL;
	bSavePB_Uni 									: BOOL; 														(*Universal*) (* Input - HMI - Save Push Button on Touchscreen*)
	bLoadPB_Uni 									: BOOL;														(*Universal*) (* Input - HMI - Load Push Button on Touchscreen*)
	bClearPB_SSER									: BOOL;
	bClearPB_SSUR									: BOOL;
	bTrackerEn										: BOOL;														(*During Tracker, it will only call arm when process completed*)
	bTrackerBasedOnPreviousTime					: BOOL;
	bMinMaxEn(*bProcessCompleteBasedMasterTime*)		: BOOL;
	bEffTimePriorityEn									: BOOL;
	bBasketTransferCallArmInterlock			: BOOL; (* Temporary -> for GPM Only*)

	(*fbGnrStationMasterController*)
	iCurrentStationAddress_Fix 							: INT;															(*Individual*) (* Input - Define current station no so that this fb know which array number to used*)
	iPreCallArmTime_Uni								: INT;															(*Universal*) (* Input - Pre-Call Arm Time, Program will call arm if the Total process timeEV Equal or Lesser than this value*)
	ARbAlternateStnEn								: ARRAY [1..iAlternateSetQty] OF BOOL;
	AR2siAlternateStn 									: ARRAY [1..iAlternateSetQty, 1..iAlternateStnQty] OF INT;

	
	
END_VAR

VAR_IN_OUT PERSISTENT

	(*fbStnSeqProcess*)
(*	DsStnSeqProInput_Ind 						: DS_StnSeqProInput;												(*Individual*) (* Input - PV of Instrument (Temperature, pressure, vacuum and etc), Signal of Sensor to allowed program under the current station status.*)
*)	DSStnSeqProcessCtrl_Ind			 		: DS_fbStnSeqProcessCtrl;											(*Individual*) (* InOut - Link with fbStnSeqProcess, so that this fb know the full status of fbStnSeqProcess and determine which action to take*)

	DsStnSeqRepStore_Ind 					: DSV2_fbStationSequenceRecipeStore; 								(*Individual*) (* InOut - HMI - The full set of DataStructure-StationSequenceRecipe should selectively display on HMI so that user can customise the recipe by choosing/configure the parameters.*)
	DsStnSubRepStore_Ind 					: DS_fbStationSubRecipeStore; 										(*Individual*) (* InOut - HMI - The full set of DataStructure-StationSubRecipe should selectively display on HMI so that user can customise the recipe by choosing/configure the parameters.*)
	DsStnSeqRepCall_Ind 						: DSV2_fbStationSequenceRecipeCall;									(*Individual*) (* InOut - Used to call StationSequenceRecipe Detail from fbStationSequenceRecipe*)
	DsStnSubRepCall_Ind 						: DS_fbStationSubRecipeCall;										(*Individual*) (* InOut - Used to call StationSubRecipe Detail from fbStationSubRecipe*)
	ARDsSSERSourceMinMaxTime_Uni						: ARRAY [1..iStnQty] OF DSV2_SSERSourceMinMaxTime;

	(*fbGnrStationMasterController*)
	ARbProductRecipeCallEn_Uni 				: ARRAY [0..iStnQty] OF BOOL;										(*Universal*) (* Output - Link with fbGnrProductRecipeMemory, Array based on Current Station No, the fbGnrProductRecipeMemory will start Read info from Memory when this bool turn on*)
	ARiProductRecipeNoCall_Uni 				: ARRAY [0..iStnQty] OF INT;										(*Universal*) (* Output - Link with fbGnrProductRecipeMemory, Array based on Current Station No, the read out from fbGnrProductRecipeMemory is based on this Product Recipe No*)
	ARiProductRecipeStepCall_Uni 				: ARRAY [0..iStnQty] OF INT;										(*Universal*) (* Output - Link with fbGnrProductRecipeMemory, Array based on Current Station No, the read out from fbGnrProductRecipeMemory is based on this Product Recipe Step No*)

	DSfbGnrProductRecipeMemoryOut_Uni 		: DSV2_fbGnrProductRecipeMemoryOut;								(*Universal*) (* Input - Link with fbGnrProductRecipeMemory, all the read out info from fbGnrProductRecipeMemory will store in this DataStucture*)

	ARbArmReady_Uni						: ARRAY [1..iArmQty] OF BOOL;										(* Universal*) (* Input  - From ArmPnpFB, This signal is used to confirm if the arm is ready and idling*)

	ARiStnNoToCalledArm_Uni					: ARRAY [0..iArmQty] OF INT; 										(*Universal*) (* Output - Link with fbArmPnP, Array based on Arm No, The Int will store which Station that calling the Arm*)
	ARDSGnrFeedArmPnpParameter_Uni		: ARRAY [0..iArmQty] OF DSV2_Gnr_CalledArmPnpParameter; 			(*Universal*) (* Output - Link with fbArmPnP, Array based on Current Station No, Arm should move based on this DataStructure Info*)

	ARDSLdBasketInfo_Uni		 			: ARRAY [0..iLdStnQty] OF DSV2_BasketInfo;								(*Input - Loading CONFIRM Basket Info*)
	ARDSUldBasketInfo_Uni		 			: ARRAY [0..iUldStnQty] OF DSV2_BasketInfo;							(*Input - Uloading CONFIRM Basket Info*)
	ARDsStnBasketInfo_Uni					: ARRAY [0..iStnQty] OF DSV2_BasketInfo;								(*Input - Station Basket Info*)



END_VAR

VAR_OUTPUT PERSISTENT
	bSaveInd_Uni 								: BOOL; 														(*Universal*) (* Output - HMI - Save Indicator on Touchscreen*)
	bLoadInd_Uni 								: BOOL; 														(*Universal*) (* Output - HMI - Load Indicator on Touchscreen*)
	bClearInd_SSER 								: BOOL;
	bClearInd_SSUR 								: BOOL;
(*	DSStnSeqProOutput_Ind 						:DS_StnSeqProOutput;											(*Individual*) (* Output - To Control Output - When process running, instrument should control by the output in this Data structure*)
*)

	bStationProcessCompleted : BOOL;
END_VAR



VAR PERSISTENT
	(*fbStnSeqProcess*)
	StnSeqProcessfb						: fbV2_StnSeqProcess;
	bStnSeqProcessStartInterlock			: BOOL;																	(*Individual*) (* Input - Interlocking to Enable the StnSeqProcess Start Signal, It might used on those station with Sliding door for close confirmation before process start*)

	(*fbGnrStationMasterController*)
	GnrStationMasterControllerfb				: fbV2_GnrStationMasterController;
	bStnSeqProcessSt						: BOOL;																(* Output - Link with fbStnSeqProcess, After Read out from fbGnrProductRecipeMemory, this fb will trigger this Bool to start the StnSeqProcess*)
	DSGnrBufferCalledArmPnpParameter 		: DSV2_Gnr_CalledArmPnpParameter;									(* Internal used, Buffer Data Structure read out from fbGnrProductRecipeMemory*)
	DSGnrBuffersPnpSequenceDescription		: STRING (99);														(* Internal used, Buffer Description read out from fbGnrProductRecipeMemory*)
	ARiPreviousStnSeqTotalProcessTime 		: ARRAY [0..iProductRecipeArrayQty] OF INT;								(* Internal used, Previous Total Process Time will save into this Array, Array based on StationSequenceNo*)
	iCallStep									: INT;																(* Internal used, to monitor the current Step so that you can indentify the error of this function block if stucked*)
	DSBasketInfo_Ind 							: DSV2_BasketInfo;														(*Individual*) (* InOut - Basket Information that comes into current station*)
	iNonStopCurrentProcessTime: INT;
END_VAR
VAR
	bLdStnConfirm: BOOL;
	bUldStnConfirm: BOOL;
	bStn1Confirm: BOOL;
	bGreaterStn1Confirm: BOOL;
	bLesserStnQtyConfirm: BOOL;
	bEqualStnQtyConfirm: BOOL;
	iTotalProcessTimeSV: INT;
	fbV2BasketInfoFinder_Ind: fbV2_BasketInfoFinder;
	iTotalProcessTimeCallForGnrStationMC: INT;
	iMasterTimeCallArmCountDownTime: INT;
	iMasterTimeBasedProcessCompleteFlag : BOOL;


	iMasterTimeBasedProcessCompleteFlagHR: BOOL;
	iProductRecipeBuffer: INT;
	bProductRecipeNoChangedFlag: BOOL;
END_VAR
VAR // added by the converter: edge detectors and wires of the graphical bodies
    _w1, _w2 : INT;
END_VAR

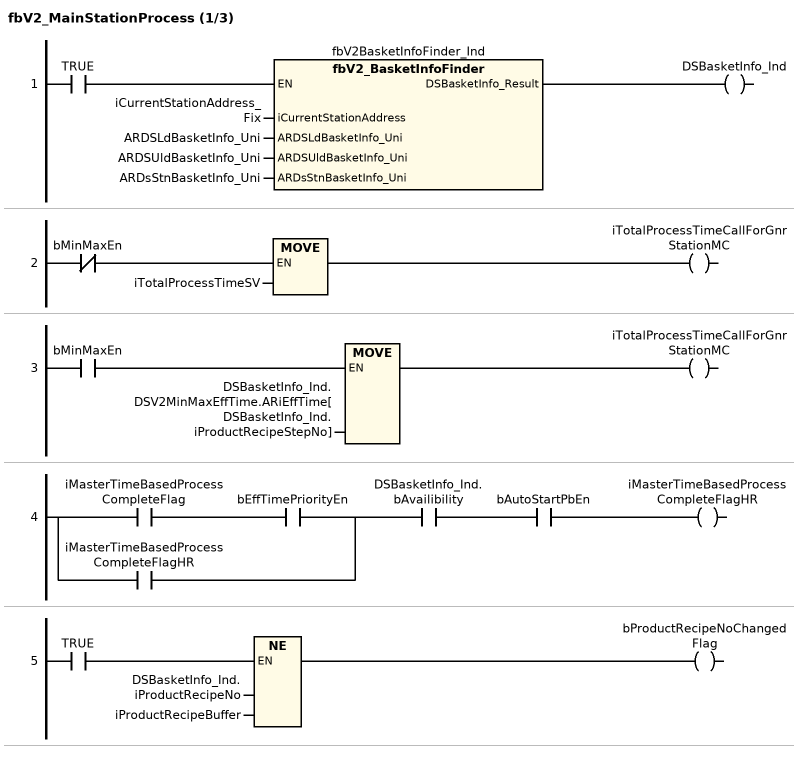
// NETWORK 1
fbV2BasketInfoFinder_Ind(
    iCurrentStationAddress := iCurrentStationAddress_Fix,
    ARDSLdBasketInfo_Uni := ARDSLdBasketInfo_Uni,
    ARDSUldBasketInfo_Uni := ARDSUldBasketInfo_Uni,
    ARDsStnBasketInfo_Uni := ARDsStnBasketInfo_Uni); // fbV2_BasketInfoFinder
DSBasketInfo_Ind := fbV2BasketInfoFinder_Ind.DSBasketInfo_Result;

// NETWORK 2
IF NOT bMinMaxEn THEN _w1 := iTotalProcessTimeSV; END_IF
iTotalProcessTimeCallForGnrStationMC := _w1;

// NETWORK 3
IF bMinMaxEn THEN
    _w2 := DSBasketInfo_Ind.DSV2MinMaxEffTime.ARiEffTime[DSBasketInfo_Ind.iProductRecipeStepNo];
END_IF
iTotalProcessTimeCallForGnrStationMC := _w2;

// NETWORK 4
iMasterTimeBasedProcessCompleteFlagHR := (iMasterTimeBasedProcessCompleteFlag AND bEffTimePriorityEn OR iMasterTimeBasedProcessCompleteFlagHR) AND DSBasketInfo_Ind.bAvailibility AND bAutoStartPbEn;

// NETWORK 5
bProductRecipeNoChangedFlag := DSBasketInfo_Ind.iProductRecipeNo <> iProductRecipeBuffer;

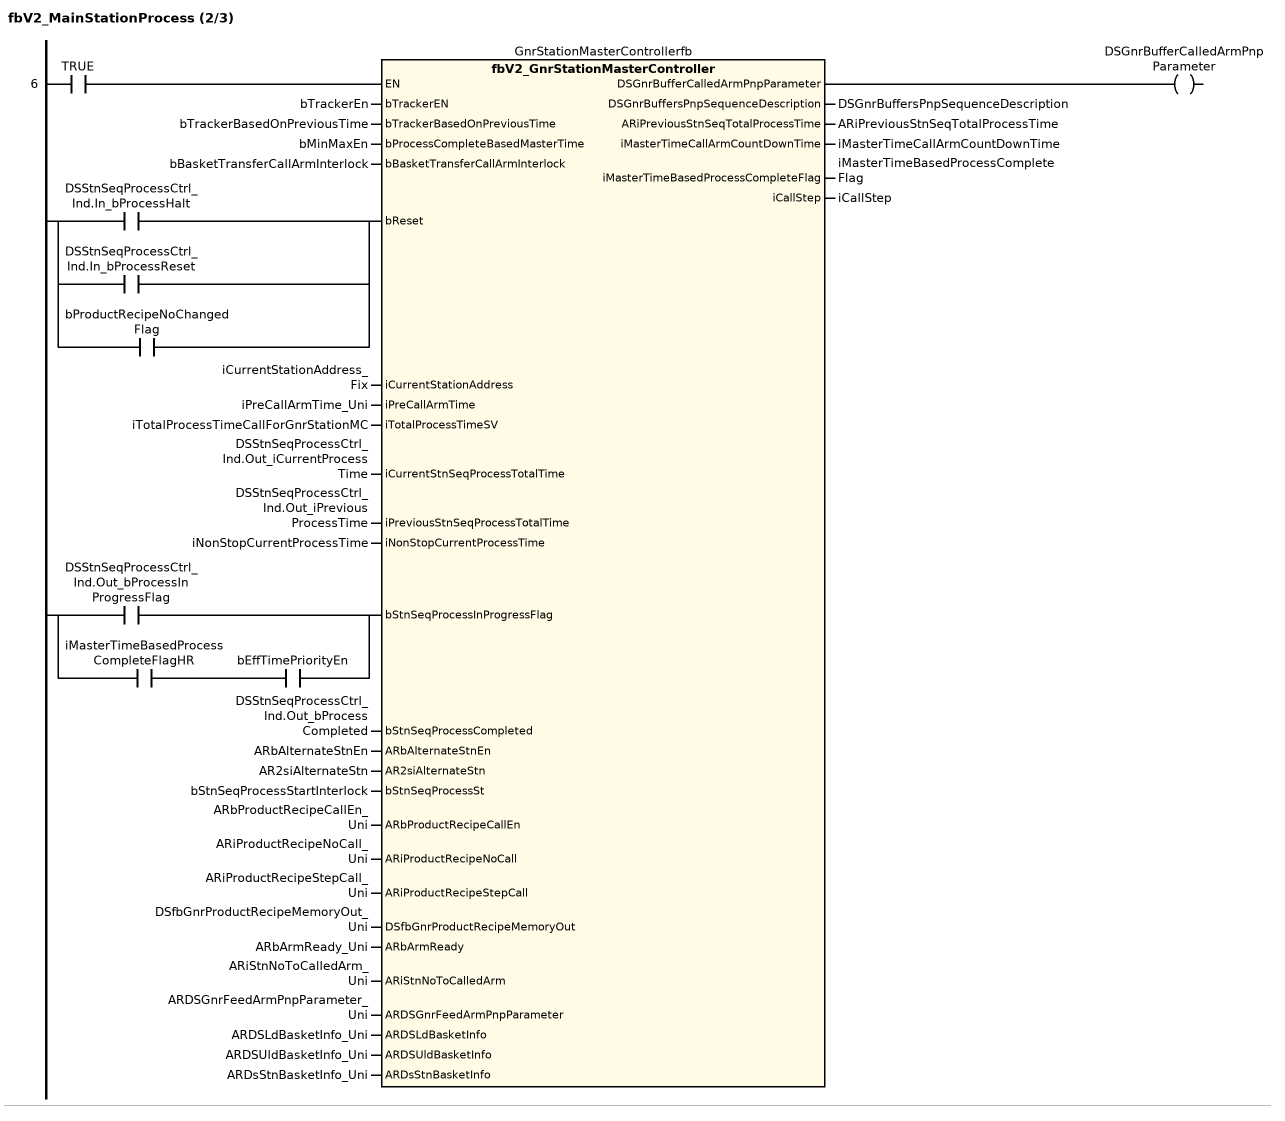
// NETWORK 6
GnrStationMasterControllerfb(
    bTrackerEN := bTrackerEn,
    bTrackerBasedOnPreviousTime := bTrackerBasedOnPreviousTime,
    bProcessCompleteBasedMasterTime := bMinMaxEn,
    bBasketTransferCallArmInterlock := bBasketTransferCallArmInterlock,
    bReset := DSStnSeqProcessCtrl_Ind.In_bProcessHalt OR DSStnSeqProcessCtrl_Ind.In_bProcessReset OR bProductRecipeNoChangedFlag,
    iCurrentStationAddress := iCurrentStationAddress_Fix,
    iPreCallArmTime := iPreCallArmTime_Uni,
    iTotalProcessTimeSV := iTotalProcessTimeCallForGnrStationMC,
    iCurrentStnSeqProcessTotalTime := DSStnSeqProcessCtrl_Ind.Out_iCurrentProcessTime,
    iPreviousStnSeqProcessTotalTime := DSStnSeqProcessCtrl_Ind.Out_iPreviousProcessTime,
    iNonStopCurrentProcessTime := iNonStopCurrentProcessTime,
    bStnSeqProcessInProgressFlag := DSStnSeqProcessCtrl_Ind.Out_bProcessInProgressFlag OR iMasterTimeBasedProcessCompleteFlagHR AND bEffTimePriorityEn,
    bStnSeqProcessCompleted := DSStnSeqProcessCtrl_Ind.Out_bProcessCompleted,
    ARbAlternateStnEn := ARbAlternateStnEn,
    AR2siAlternateStn := AR2siAlternateStn,
    bStnSeqProcessSt := bStnSeqProcessStartInterlock,
    ARbProductRecipeCallEn := ARbProductRecipeCallEn_Uni,
    ARiProductRecipeNoCall := ARiProductRecipeNoCall_Uni,
    ARiProductRecipeStepCall := ARiProductRecipeStepCall_Uni,
    DSfbGnrProductRecipeMemoryOut := DSfbGnrProductRecipeMemoryOut_Uni,
    ARbArmReady := ARbArmReady_Uni,
    ARiStnNoToCalledArm := ARiStnNoToCalledArm_Uni,
    ARDSGnrFeedArmPnpParameter := ARDSGnrFeedArmPnpParameter_Uni,
    ARDSLdBasketInfo := ARDSLdBasketInfo_Uni,
    ARDSUldBasketInfo := ARDSUldBasketInfo_Uni,
    ARDsStnBasketInfo := ARDsStnBasketInfo_Uni,
    DSGnrBuffersPnpSequenceDescription => DSGnrBuffersPnpSequenceDescription,
    ARiPreviousStnSeqTotalProcessTime => ARiPreviousStnSeqTotalProcessTime,
    iMasterTimeCallArmCountDownTime => iMasterTimeCallArmCountDownTime,
    iMasterTimeBasedProcessCompleteFlag => iMasterTimeBasedProcessCompleteFlag,
    iCallStep => iCallStep); // fbV2_GnrStationMasterController
DSGnrBufferCalledArmPnpParameter := GnrStationMasterControllerfb.DSGnrBufferCalledArmPnpParameter;

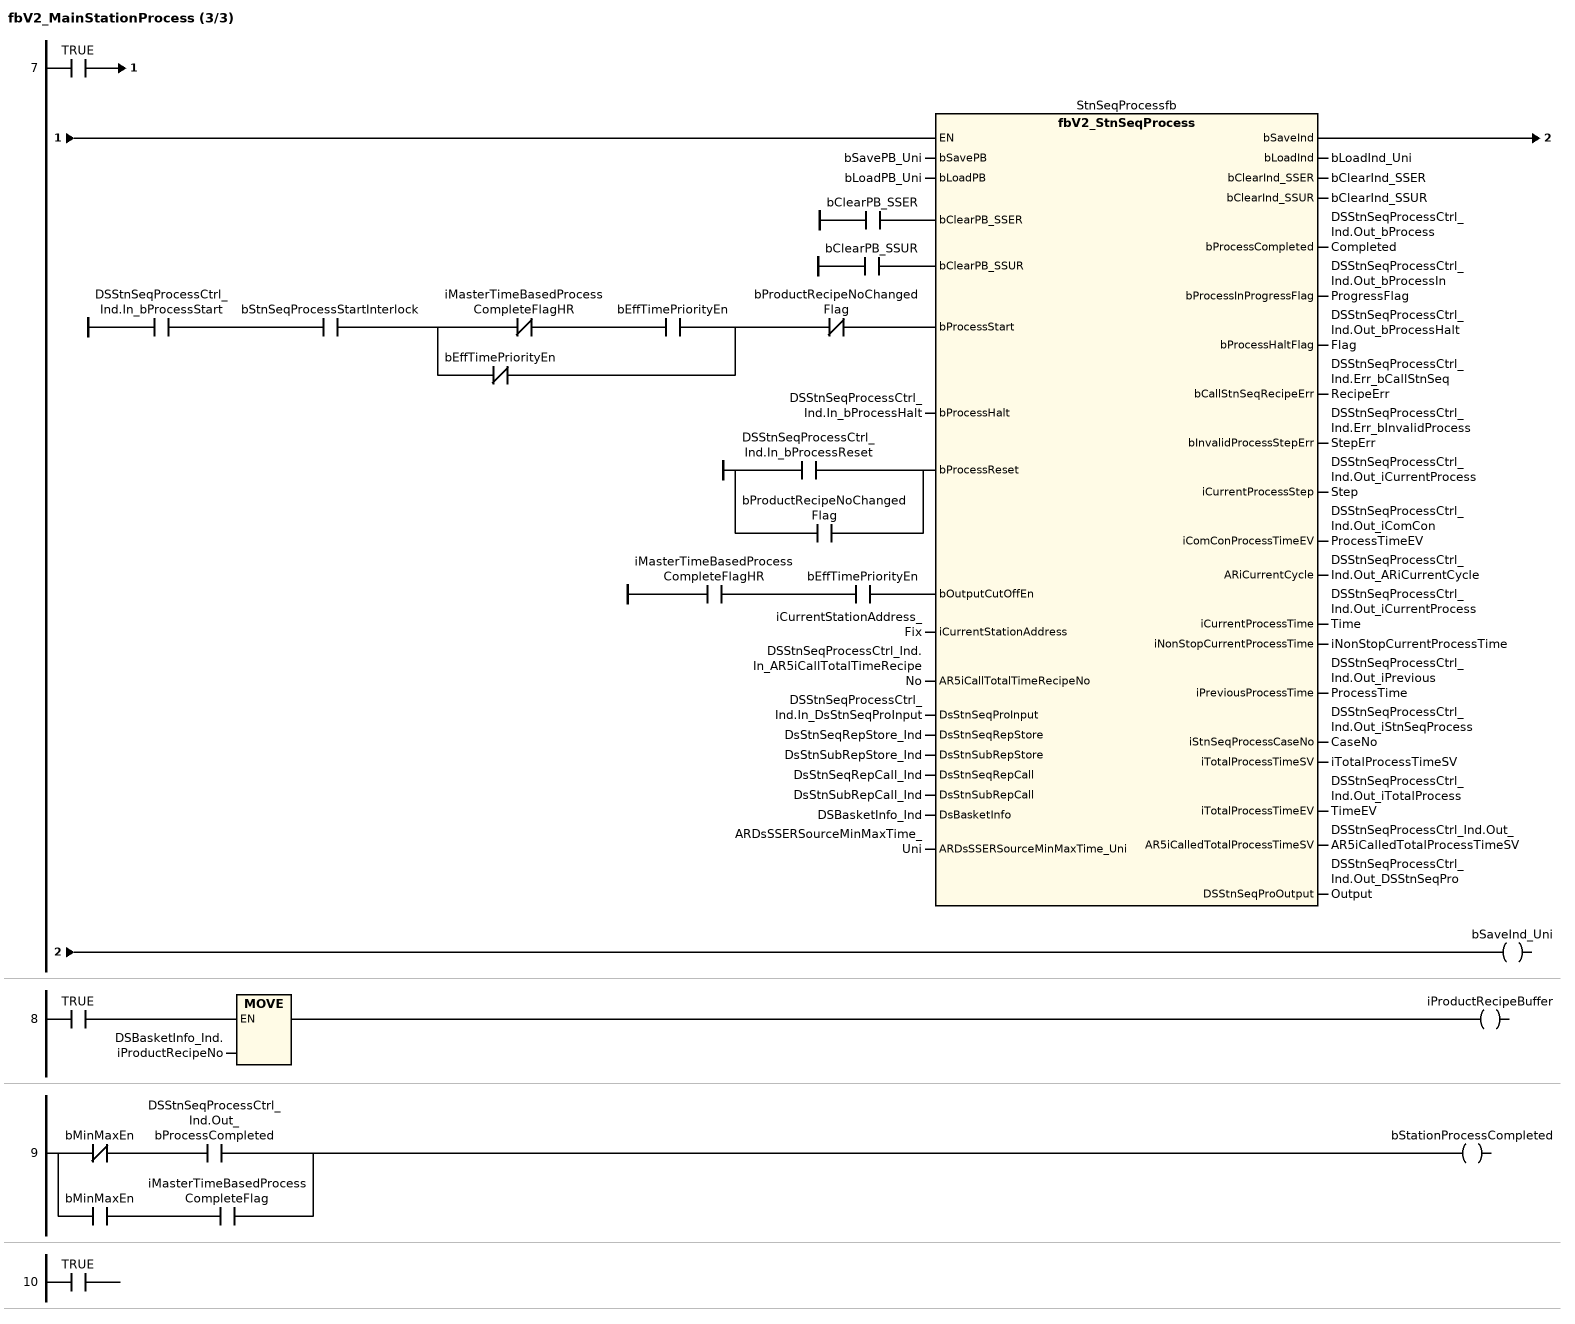
// NETWORK 7
StnSeqProcessfb(
    bSavePB := bSavePB_Uni,
    bLoadPB := bLoadPB_Uni,
    bClearPB_SSER := bClearPB_SSER,
    bClearPB_SSUR := bClearPB_SSUR,
    bProcessStart := ((DSStnSeqProcessCtrl_Ind.In_bProcessStart AND bStnSeqProcessStartInterlock) AND (NOT iMasterTimeBasedProcessCompleteFlagHR AND bEffTimePriorityEn OR NOT bEffTimePriorityEn)) AND NOT bProductRecipeNoChangedFlag,
    bProcessHalt := DSStnSeqProcessCtrl_Ind.In_bProcessHalt,
    bProcessReset := DSStnSeqProcessCtrl_Ind.In_bProcessReset OR bProductRecipeNoChangedFlag,
    bOutputCutOffEn := iMasterTimeBasedProcessCompleteFlagHR AND bEffTimePriorityEn,
    iCurrentStationAddress := iCurrentStationAddress_Fix,
    AR5iCallTotalTimeRecipeNo := DSStnSeqProcessCtrl_Ind.In_AR5iCallTotalTimeRecipeNo,
    DsStnSeqProInput := DSStnSeqProcessCtrl_Ind.In_DsStnSeqProInput,
    DsStnSeqRepStore := DsStnSeqRepStore_Ind,
    DsStnSubRepStore := DsStnSubRepStore_Ind,
    DsStnSeqRepCall := DsStnSeqRepCall_Ind,
    DsStnSubRepCall := DsStnSubRepCall_Ind,
    DsBasketInfo := DSBasketInfo_Ind,
    ARDsSSERSourceMinMaxTime_Uni := ARDsSSERSourceMinMaxTime_Uni,
    bLoadInd => bLoadInd_Uni,
    bClearInd_SSER => bClearInd_SSER,
    bClearInd_SSUR => bClearInd_SSUR,
    bProcessCompleted => DSStnSeqProcessCtrl_Ind.Out_bProcessCompleted,
    bProcessInProgressFlag => DSStnSeqProcessCtrl_Ind.Out_bProcessInProgressFlag,
    bProcessHaltFlag => DSStnSeqProcessCtrl_Ind.Out_bProcessHaltFlag,
    bCallStnSeqRecipeErr => DSStnSeqProcessCtrl_Ind.Err_bCallStnSeqRecipeErr,
    bInvalidProcessStepErr => DSStnSeqProcessCtrl_Ind.Err_bInvalidProcessStepErr,
    iCurrentProcessStep => DSStnSeqProcessCtrl_Ind.Out_iCurrentProcessStep,
    iComConProcessTimeEV => DSStnSeqProcessCtrl_Ind.Out_iComConProcessTimeEV,
    ARiCurrentCycle => DSStnSeqProcessCtrl_Ind.Out_ARiCurrentCycle,
    iCurrentProcessTime => DSStnSeqProcessCtrl_Ind.Out_iCurrentProcessTime,
    iNonStopCurrentProcessTime => iNonStopCurrentProcessTime,
    iPreviousProcessTime => DSStnSeqProcessCtrl_Ind.Out_iPreviousProcessTime,
    iStnSeqProcessCaseNo => DSStnSeqProcessCtrl_Ind.Out_iStnSeqProcessCaseNo,
    iTotalProcessTimeSV => iTotalProcessTimeSV,
    iTotalProcessTimeEV => DSStnSeqProcessCtrl_Ind.Out_iTotalProcessTimeEV,
    AR5iCalledTotalProcessTimeSV => DSStnSeqProcessCtrl_Ind.Out_AR5iCalledTotalProcessTimeSV,
    DSStnSeqProOutput => DSStnSeqProcessCtrl_Ind.Out_DSStnSeqProOutput); // fbV2_StnSeqProcess
bSaveInd_Uni := StnSeqProcessfb.bSaveInd;

// NETWORK 8
iProductRecipeBuffer := DSBasketInfo_Ind.iProductRecipeNo;

// NETWORK 9
bStationProcessCompleted := NOT bMinMaxEn AND DSStnSeqProcessCtrl_Ind.Out_bProcessCompleted OR bMinMaxEn AND iMasterTimeBasedProcessCompleteFlag;

// NETWORK 10

END_FUNCTION_BLOCK

// ---- FBs/B_JKS_NewFB_V2/FBP-Memory_Sub/fbV2_StnSeqProcess.TcPOU
FUNCTION_BLOCK fbV2_StnSeqProcess

VAR_INPUT
	bSavePB 							: BOOL; 									(* Input - HMI - Save Push Button on Touchscreen*)
	bLoadPB 							: BOOL;									(* Input - HMI - Load Push Button on Touchscreen*)
	bClearPB_SSER						: BOOL;
	bClearPB_SSUR						: BOOL;
	bProcessStart 					: BOOL;									(* Input - To Trigger process start - Pulse Signal*)
	bProcessHalt						: BOOL;									(* Input - To Trigger Process Halt/Pause*)
	bProcessReset 					: BOOL;									(* Input - To Process Reset/Initialization*)
	bOutputCutOffEn 					: BOOL;									(* Input - To Process Reset/Initialization*)

	iCurrentStationAddress 					: INT;															(* Input - Define current station no so that this fb know which array number to used*)
	AR5iCallTotalTimeRecipeNo 	: ARRAY [1..5] OF INT;						(* Input - It can accept concurrently 5 different Recipe No, with the reference of Recipe No, it will trace out the total time of that particular recipe by output to AR5iCalledTotalProcessTimeSV*)
	DsStnSeqProInput 				: DS_StnSeqProInput;						(* Input - PV of Instrument (Temperature, pressure, vacuum and etc), Signal of Sensor to allowed program under the current station status.*)

	
END_VAR

VAR_IN_OUT PERSISTENT
	DsStnSeqRepStore 				: DSV2_fbStationSequenceRecipeStore; 	(* InOut - HMI - The full set of DataStructure-StationSequenceRecipe should selectively display on HMI so that user can customise the recipe by choosing/configure the parameters.*)
	DsStnSubRepStore 				: DS_fbStationSubRecipeStore; 			(* InOut - HMI - The full set of DataStructure-StationSubRecipe should selectively display on HMI so that user can customise the recipe by choosing/configure the parameters.*)

	DsStnSeqRepCall 				: DSV2_fbStationSequenceRecipeCall;		(* InOut - Used to call StationSequenceRecipe Detail from fbStationSequenceRecipe*)
	DsStnSubRepCall 				: DS_fbStationSubRecipeCall;			(* InOut - Used to call StationSubRecipe Detail from fbStationSubRecipe*)

	DsBasketInfo 						: DSV2_BasketInfo;							(* InOut - Basket Information that comes into current station*)
	ARDsSSERSourceMinMaxTime_Uni						: ARRAY [1..iStnQty] OF DSV2_SSERSourceMinMaxTime;

END_VAR

VAR_OUTPUT PERSISTENT
	bSaveInd 							: BOOL; 												(* Output - HMI - Save Indicator on Touchscreen*)
	bLoadInd 							: BOOL; 												(* Output - HMI - Load Indicator on Touchscreen*)
	bClearInd_SSER						: BOOL;
	bClearInd_SSUR						: BOOL;
	bProcessCompleted 				: BOOL;												(* Output - Bool will turn on once the full process completed*)
	bProcessInProgressFlag 		: BOOL;												(* Output - Bool will turn on once the process Start, will off when process completed*)
	bProcessHaltFlag					: BOOL;												(* Output - Bool will turn on during Process Halt/Paused*)

	bCallStnSeqRecipeErr			: BOOL;												(* Output - Error - Bool will turn on when it face problem during StnSeqRecipe Called process*)
	bInvalidProcessStepErr			: BOOL;												(* Output - Error - Bool will turn on when it found the given step number is Invalid*)
	iCurrentProcessStep 				: INT;													(* Internal used, to monitor the current Step so that you can indentify the error of this function block if stucked*)
	iComConProcessTimeEV		: INT;													(* Output - HMI - Timer Elapse Value (DownCounting) of current process steps*)
	ARiCurrentCycle 					: ARRAY [1..iProductRecipeStepArrayQty] OF INT;	(* Output - HMI - Array based on Steps No, Current Cycle No on that particular Steps*)
	iCurrentProcessTime 			: INT; 													(* Output - Current Process Time (Current Steps) Since Start (UpCounting)*)
	iNonStopCurrentProcessTime: INT;
	iPreviousProcessTime 			: INT; 													(* Output - Previous Total Process Time*)
	iStnSeqProcessCaseNo			: INT;		 											(* Internal used, to monitor the current Step so that you can indentify the error of this function block if stucked*)
	iTotalProcessTimeSV: 			INT;

	iTotalProcessTimeEV				: INT; 													(* Output - Total Process Elapse Time (DownCounting) (Based Total Time) *)
	AR5iCalledTotalProcessTimeSV	: ARRAY [1..5] OF INT;									(* Output -  It can accept concurrently 5 different Recipe Total Time based on the Recipe Number defined in AR5iCallTotalTimeRecipeNo*)
	DSStnSeqProOutput 				:DS_StnSeqProOutput;								(* Output - To Control Output - When process running, instrument should control by the output in this Data structure*)
END_VAR
VAR
	DsStnSeqRepCallEmpty 				: DSV2_fbStationSequenceRecipeCall;		(* Empty*)
	DsStnSubRepCallEmpty 				: DS_fbStationSubRecipeCall;			(*Empty*)

	rebProcessStart: R_TRIG;


	bCallStnSeqSubProEn: BOOL;

	bStCon11BelowTargetVacuumLevel : BOOL;
	bStCon12AboveTargetVacuumLevel : BOOL;
	bStCon13BelowTargetPressureLevel : BOOL;
	bStCon14AboveTargetPressureLevel : BOOL;
	bStCon15BelowTargetProTankTempLevel : BOOL;
	bStCon16AboveTargetProTankTempLevel : BOOL;
	bStCon17BelowTargetSubTankTempLevel : BOOL;
	bStCon18AboveTargetSubTankTempLevel : BOOL;

	bComCon11BelowTargetVacuumLevel : BOOL;
	bComCon12AboveTargetVacuumLevel : BOOL;
	bComCon13BelowTargetPressureLevel : BOOL;
	bComCon14AboveTargetPressureLevel : BOOL;
	bComCon15BelowTargetProTankTempLevel : BOOL;
	bComCon16AboveTargetProTankTempLevel : BOOL;
	bComCon17BelowTargetSubTankTempLevel : BOOL;
	bComCon18AboveTargetSubTankTempLevel : BOOL;

	tProcess1secClockPulse: TON;
	retProcess1secClockPulse: R_TRIG;
	rebProcessCompleted: R_TRIG;
	ClearFL: INT;
	iCurrentProcessStepBuffer: INT;
	rebInvalidProcessStepErr: R_TRIG;
	rebStnSeqSubCallCompleted: R_TRIG;
	rebCallStnSeqRecipeErr: R_TRIG;
	rebCallStnSubRecipeErr: R_TRIG;
	tStartProcess1secClockPulse: TON;
	retStartProcess1secClockPulse: R_TRIG;
	bTempCallCompleted: BOOL;
	bTempInvalidProcessStepErr: BOOL;
	bTempCallStnSeqRecipeErr: BOOL;
	bTempCallStnSubRecipeErr: BOOL;
	sTempsSubDescription: STRING(50);
	DsTempSubRecipeMemory: DS_SubRecipeMemory;
	iTempSeqStep: INT;
	bTempInvalidProcessStepErrPls: BOOL;
	rebProcessHalt: R_TRIG;
	febProcessHalt: F_TRIG;
	iTPTFL: INT;
	iEndStep: INT;
	iCTPTFL: INT;
	bEndStep: BOOL;

	iCallTotalTimeMFL: INT;
	iCallTotalTimeSFL: INT;
	bCallTotalTimeEndStep: BOOL;
	iCalculateMFL: INT;
	iCalculateSFL: INT;

END_VAR

VAR PERSISTENT
	fbStationSequenceRecipefb: fbV2_StationSequenceRecipe;
	fbStationSubRecipefb: fbStationSubRecipe;
	StationfbCallStnSeqSubPro: fbV2_CallStnSeqSubPro;
	bStartConditionPassed: BOOL;
	bCompleteConditionPassed: BOOL;
	bStationProcessTimerComplete: BOOL;
	iComConProcessTime: INT;
	ARiTotalTimeSV: ARRAY [1..IStationSubRecipeArrayQty] OF INT;
	AR2SiTimeOptimiseTotalTimeSV: ARRAY [1..5, 1..IStationSubRecipeArrayQty] OF INT;
	iTotalProcessTimeEVInt: INT;

END_VAR





(*
(*[][][][][][][][][][][][][][][][][][][][][][][][][][][][][][][][][][][][][][][][][][][][][][][][][][][][][][][][][][][][][][][][][][][][][][][][]-Original for FB StnSeqProcess Backup-[][][][][][][][][][][][][][][][][][][][][][][][][][][][][][][][][][][][][][][][][][][][][][][][][][][][][][][][][][][][][][][][][][][][][][][][]*)

VAR_INPUT
	bProcessStart : BOOL;
	bProcessHalt: BOOL;
	bProcessReset : BOOL;
	DsStnSeqProInput :DS_StnSeqProInput;

END_VAR

